	IF NOT Busy                                         	
	THEN                                                	
		IF ItpReadRParamsEx.bExecute                    	
		THEN                                            	
			Error											:=	ItpReadRParamsEx.bErr;
			ErrorId											:= ItpReadRParamsEx.nErrId;
		END_IF                          					
		IF NOT Execute                  					
		THEN                            	            	
			MemFnc											:= -1;
			ItpReadRParamsEx(bExecute := FALSE , sNciToPlc:= rNCIRef.NciToPlc);
		END_IF
	END_IF
	
	read													:= Busy;
END_METHOD

METHOD PUBLIC write : BOOL //Return value = TRUE if busy
//required parameter
//pAddr
//Index
//Count
//rNCIRef
VAR_INPUT
	Execute													:	BOOL;
END_VAR
	MemFnc 													:= FNC_WRITE;
	THIS^.Execute											:= Execute;

IF NOT __ISVALIDREF(rNCIRef) OR pAddr = 0 
THEN
	Busy													:= NOT Error;
	ErrorId													:= E_adsErr.DEVICE_INVALIDPARM;
	Error													:= TRUE;
	Done													:= FALSE;
	MemFnc													:= SEL(Execute , -1 ,MemFnc); 
	RETURN;
END_IF

	IF Execute
	THEN
		Error												:=	FALSE;
		ErrorId												:= 0;
		ItpWriteRParamsEx.bExecute 							:= TRUE;
	ELSIF NOT ItpWriteRParamsEx.bBusy   					
	THEN                                					
		Error												:=	FALSE;
		ErrorId												:= 0;
		ItpWriteRParamsEx.bExecute 							:= FALSE;

	END_IF

	ItpWriteRParamsEx(
		bExecute	:= ,
		pAddr		:= pAddr,
		nIndex		:= Index,
		nCount		:= Count,
		tTimeOut	:= ,
		sNciToPlc	:= rNCIRef.NciToPlc,
		bBusy		=> Busy,
		bErr		=> ,
		nErrId		=> );

	Done													:= NOT ItpWriteRParamsEx.bBusy
																AND NOT ItpWriteRParamsEx.bErr
																AND ItpWriteRParamsEx.bExecute;
                                        					
	IF NOT Busy
	THEN
		IF ItpWriteRParamsEx.bExecute
		THEN
			Error											:=	ItpWriteRParamsEx.bErr;
			ErrorId											:= ItpWriteRParamsEx.nErrId;
		END_IF                          					
		IF NOT Execute                  					
		THEN                            	
			MemFnc											:= -1;
			ItpWriteRParamsEx(bExecute := FALSE, sNciToPlc:= rNCIRef.NciToPlc);
		END_IF
	END_IF
	
	write													:= Busy;
END_METHOD

END_FUNCTION_BLOCK

// POUs/Motion/TF5100-NCI/NciChannel
{attribute 'no_check'}
FUNCTION_BLOCK NciChannel EXTENDS NCI_REF
VAR_INPUT
	Admin													:	NciAdmin;
	grp														:	NciGrp;
	Itp														:	NciItp;
	motion													:	NciMotion;
                        								   
	MFnc													: 	NciMFnc;
	RPara													:	NciReadWriteRParam;
                        								      
	Event													:	NciEventHandling;
                        	
END_VAR                 	
VAR_OUTPUT              	
	ErrHdl													:	ERROR_HDL;
END_VAR
VAR
END_VAR

	(* NCI Control											*)
	(********************************************************)

(********************************************************************************)
(* error event ctrl																*)
(********************************************************************************)
	Event(
		Enable			:= ,
		ConfirmTrig		:= NOT Errhdl.flag AND Event.Status.31 OR Admin.ResetAdmin,
		Name			:= ErrHdl.fnc,
		SourceId		:= (* Default *) ,
		rNci			:= THIS^,
		ErrorId			:= TO_UDINT(ErrHdl.Id),
		Status			=> );
		
	(* Reset FB errors by reset flag *)
	(* currently not in use, call _Resetting via state machine to reset Fb errors by setting Execute to FALSE 
	IF Admin.Reset
	THEN
		grp.Execute											:= grp.Execute AND NOT grp.Error;
		itp.Execute											:= itp.Execute AND NOT itp.Error;
		Motion.Execute										:= Motion.Execute AND NOT Motion.Error;
		RPara.Execute										:= RPara.Execute AND NOT RPara.Error;
	END_IF
	*)
	
(********************************************************************************)
(* work admin ctrl																*)
(********************************************************************************)
	admin(
		ResetAdmin					:= ,
		Enable					:= ,
		EStop					:= ,
		SingleBlockMode			:= , 
		InSingleBlockTrigNext	:= , 
		GrpCnfg					:= ,
		Override				:= ,
		SpindleOvr				:= ,	
		rNCIRef					:= THIS^,
		InGroup					=> ,
		Busy					=> ,
		Done					=> ,
		Error					=> ,
		ErrorID					=> ,
		ErrorText				=> );

(********************************************************************************)
(* work group ctrl																*)
(********************************************************************************)
	grp(
		Execute				:= ,
		Fnc					:= ,
		XAxisId				:= ,
		YAxisId				:= ,
		ZAxisId				:= ,
		Q1AxisId			:= ,
		Q2AxisId			:= ,
		Q3AxisId			:= ,
		Q4AxisId			:= ,
		Q5AxisId			:= ,
		AxisIndex			:= ,
		rNCIRef				:= THIS^, 
		Busy				=> ,
		Done				=> ,
		Error				=> ,
		ErrorID				=> ,
		ErrorText			=> );

(********************************************************************************)
(* work interpolation ctrl														*)
(********************************************************************************)
	Itp(
		Execute				:= ,
		Fnc					:= ,
		Prg					:= ,
		rTable				:= ,
		rNCIRef				:= THIS^,
		StartPrgAfterLoading:= , 
		LogFeederEntries	:= ,
		Busy				=> ,
		Done				=> ,
		Error				=> ,
		ErrorID				=> ,
		ErrorText			=> );


(********************************************************************************)
(* work motion ctrl																*)
(********************************************************************************)
	motion(
		Execute						:= ,
		Fnc							:= ,
		rNCIRef						:= THIS^,
		FNC_ESTOP					=> ,
		FNC_STEP_ON					=> ,
		FNC_ENABLE_FEEDER_BACKUP	=> ,
		FNC_DISABLE_FEEDER_BACKUP	=> ,
		FNC_RETRACE_FWD				=> ,
		FNC_RETRACE_BWD				=> ,
		Busy						=> ,
		Done						=> ,
		Error						=> ,
		ErrorId						=> ,
		ErrorText					=> );

(********************************************************************************)
(* work R rarameter ctrl														*)
(********************************************************************************)
	RPara(
		Execute						:= ,
		Fnc							:= ,
		pAddr						:= ,
		Index						:= ,
		Count						:= ,
		rNCIRef						:= THIS^,
		Done						=> ,
		Busy						=> ,
		Error						=> ,
		ErrorId						=> );

(********************************************************************************)
(* work M function  ctrl														*)
(********************************************************************************)
	MFnc(
		ConfirmHsk					:= ,
		FastMFuncReset				:= ,
		FastMFuncNo					:= ,
		rNCIRef						:= THIS^);

(********************************************************************************)
(* collect errors																*)
(********************************************************************************)
	IF Admin.Error
	THEN
		ErrHdl.flag											:= Admin.Error;
		ErrHdl.id											:= UDINT_TO_DINT(Admin.ErrorID);
		ErrHdl.fnc											:= 'NciAdmin';
		ErrHdl.text											:= Admin.ErrorText;
                        									
	ELSIF grp.Error     									
	THEN                									
		ErrHdl.flag											:= grp.Error;
		ErrHdl.id											:= UDINT_TO_DINT(grp.ErrorID);
		ErrHdl.fnc											:= 'NciGrp';
		ErrHdl.text											:= grp.ErrorText;
                        									
	ELSIF itp.Error     									
	THEN                									
		ErrHdl.flag											:= Itp.Error;
		ErrHdl.id											:= UDINT_TO_DINT(Itp.ErrorID);
		ErrHdl.fnc											:= 'NciItp';
		ErrHdl.text											:= Itp.ErrorText;
                        									
	ELSIF motion.Error  									
	THEN                									
		ErrHdl.flag											:= motion.Error;
		ErrHdl.id											:= UDINT_TO_DINT(motion.ErrorID);
		ErrHdl.fnc											:= 'NciMotion';
		ErrHdl.text											:= motion.ErrorText;
		
	ELSIF RPara.Error  									
	THEN                									
		ErrHdl.flag											:= RPara.Error;
		ErrHdl.id											:= UDINT_TO_DINT(RPara.ErrorID);
		ErrHdl.fnc											:= 'RPara';
		ErrHdl.text											:= CONCAT('Error RPara id: ',  UDINT_TO_STRING(RPara.Errorid));
	ELSE
		ErrHdl.Reset();
	END_IF
(******************************************************************************)

METHOD PUBLIC noAction : BOOL
VAR_INPUT
END_VAR
grp.Execute													:= FALSE;
itp.Execute													:= FALSE;
Motion.Execute												:= FALSE;
RPara.Execute												:= FALSE;

NoAction 													:= NOT Grp.Busy and not Itp.Busy and not Motion.Busy and not RPara.Busy;
END_METHOD

METHOD reset : Bool
VAR_INPUT
END_VAR
NoAction();
reset 			:= ErrHdl.flag OR Admin.reset(FALSE);
Event.confirm();
END_METHOD

END_FUNCTION_BLOCK

// POUs/Motion/TF511x-KIN/01_Main/KIN_REF
//Kinematic group ref - call ReadStatus cyclic
FUNCTION_BLOCK KIN_REF
VAR_INPUT
	PlcToNci										AT %Q*	:	PLCTONC_NCICHANNEL_REF;
END_VAR                     						
VAR_OUTPUT                  						
	NciToPlc										AT %I*	:	NCTOPLC_NCICHANNEL_REF;
                            						
	ChnOperationState										:	E_KINSTATUS := 0;
	CartesianModeON											:	BOOL := FALSE;
	                                					
(* ChnState ***************************)
	IsKinematicChn											:	BOOL := FALSE;
	                                					
	AxList													: ST_KinAxes;
END_VAR
VAR
END_VAR

;

METHOD PUBLIC readStatus : booL;
VAR_INPUT
END_VAR
(* Kin Channel State *********************************************************)
	F_KinGetAcsMcsAxisIds(AxList,NciToPlc);
	
	ChnOperationState 										:= TO_INT(F_KinGetChnOperationState(NciToPlc));

	CartesianModeON											:= NciToPlc.AcsAxisIDs[0] <> 0 AND NciToPlc.AcsAxisIDs[1] <> 0;
	
	IsKinematicChn											:= NciToPlc.ChnState.1;

	readStatus												:= TRUE;
(*****************************************************************************)
END_METHOD

END_FUNCTION_BLOCK

// POUs/Motion/TF511x-KIN/01_Main/KinAdmin
//Kinematic group administration - Enable/Disable/Reset group
//based on TF511x - Tc2_NcKinematicTransformation
//ACS - Axis coordinate system => Robot motors M1-Mx 
//MCS - Machine coordinate system >= Cartesian Axis X,Y,Z,Rx,Ry,Rz (A,B,C) 
FUNCTION_BLOCK KinAdmin
VAR_INPUT
	ResetTrig												:	BOOL := FALSE;
	Enable													:	BOOL := FALSE; (* TRUE = Build Group , FALSE = Reconfig Group *)
	Override												:	LREAL	:= 0.0;
	ItpChannelId 											: 	UDINT := 0; (* Bei 0 wirtd der ITP Kanal nicht resetet *)
	AxesList												: 	ST_KinAxes;
	rKINRef													:	REFERENCE TO KIN_REF := 0;
END_VAR
VAR_IN_OUT
END_VAR
VAR_OUTPUT
	Busy													:	BOOL;
	Done													:	BOOL;
	Error													:	BOOL;
{attribute 'displaymode':='hex'}
	ErrorId													:	UDINT;
	ErrorText												:	STRING(40);
END_VAR
VAR
(* cache **************************************************************************)
	MemDone													:	BOOL;
	MemFnc													:	INT := 1;
	                        								
(* MC-functonblock instances *******************************************************)
	ResetKinGroup											: 	FB_KinResetGroup ;
	ConfigKinGroup											:	FB_KinConfigGroup  ;

(* Dummy Speicher **********************************************************)
	OK 														: BOOL;
END_VAR

	(* Kinematic group administration										*)
	(************************************************************************)

(* aborting function-block call if pointer is not valid ****************************************)
IF NOT __ISVALIDREF(rKINRef) 
THEN
	Busy													:= NOT Error;
	ErrorId													:= E_AdsErr.DEVICE_INVALIDPARM;
	Error													:= TRUE;
	Done													:= FALSE;
	ErrorText												:= 'Reference to rKINRef invalid (0)';
	RETURN;
END_IF

(* reading axis-status from NCtoPLC-channel ***************************************************)
	rKINRef.readStatus();

(* accepting setvalue-barrier e.g. for hardware limit switch **********************************)
	rKINRef.PlcToNci.ChnAxesOvr 							:= LREAL_TO_DWORD(LIMIT(0.0,Override,100.0) * 10000.0 );

(* ctrl programm ******************************************************************************)
	ConfigKinGroup.bExecute									:=	NOT ConfigKinGroup.bBusy
																AND(
																Enable
																AND NOT ConfigKinGroup.bCartesianMode
																OR
																NOT Enable
																AND ConfigKinGroup.bCartesianMode);

	IF ConfigKinGroup.bExecute
	THEN
		ConfigKinGroup.bCartesianMode						:= Enable;
	END_IF

	ConfigKinGroup(
		bExecute		:= ,
		bCartesianMode	:= ,
		stAxesList		:= AxesList,
		stKinRefIn		:= rKinRef.NciToPlc,
		bBusy			=> ,
		bDone			=> ,
		bError			=> ,
		nErrorId		=> );

(* Reset Grp ****************************************************************)
	IF Memfnc < 0
	THEN
		IF ResetTrig
		THEN
			reset(Execute:= TRUE);
			MemFnc											:= 1;
		END_IF
	ELSIF NOT reset(Execute:= ResetTrig)
	THEN
		MemFnc												:= -1;
	END_IF

(******************************************************************************)
(* Ctrl Status 																					*)
(******************************************************************************)
	Busy						:= ResetKinGroup.bBusy OR ConfigKinGroup.bBusy;
	
	IF Busy
	THEN
		Error												:= FALSE;
		ErrorId												:= 0;
		ErrorText											:= '';
	ELSIF ConfigKinGroup.bError
	THEN
		Error												:= TRUE;
		ErrorId												:= ConfigKinGroup.nErrorID;
		ErrorText											:= CONCAT('ConfigKinGroup ErrorId: ', UDINT_TO_STRING(Errorid));
	ELSIF ResetKinGroup.bExecute
		AND ResetKinGroup.bError
	THEN
		Error												:= TRUE;
		ErrorId												:= ResetKinGroup.nErrorID;
		ErrorText											:= CONCAT('ResetKinGroup ErrorId: ', UDINT_TO_STRING(Errorid));
	ELSIF rKINRef.NciToPlc.ErrorCode <> 0
	THEN
		Error												:= TRUE;
		ErrorId												:= rKINRef.NciToPlc.ErrorCode;
		ErrorText											:= CONCAT('KIN Grp ErrorId: ', UDINT_TO_STRING(Errorid));
	ELSE
		Error												:= FALSE;
		ErrorId												:= 0;
		ErrorText											:= '';
	END_IF

	IF ResetKinGroup.bDone
		OR ConfigKinGroup.bDone
	THEN
		MemDone												:= TRUE;
	END_IF

	Done													:= NOT Busy AND MemDone;

	IF done
	THEN
		MemDone												:= FALSE;
	END_IF

(**************************************************************************************************)

METHOD PUBLIC reset : BOOL //Return value = TRUE if busy
//required parameter
//rKinRef
//ItpChannelId
//AxesList
VAR_INPUT
	Execute													:	BOOL;
END_VAR
IF NOT __ISVALIDREF(rKINRef) THEN
	Busy													:= NOT Error;
	ErrorId													:=E_AdsErr.DEVICE_INVALIDPARM;
	Error													:= TRUE;
	Done													:= FALSE;
	ErrorText												:= 'Reference to rKINRef  invalid (0)';
	RETURN;
END_IF

	IF Execute
	THEN
		Error												:=	FALSE;
		ErrorId												:= 0;
		ResetKinGroup.bExecute 								:= rKinRef.NciToPlc.ErrorCode <> 0;
	ELSIF NOT ResetKinGroup.bBusy
	THEN
		Error												:=	FALSE;
		ErrorId												:= 0;
		ResetKinGroup.bExecute 								:= FALSE;

	END_IF

	ResetKinGroup(
		bExecute		:= ,
		nItpChannelId	:= ItpChannelId,
		stKinRefIn		:= rKinRef.NciToPlc,
		stAxesList		:= AxesList,
		bBusy			=> Busy,
		bDone			=> ,
		bError			=> ,
		nErrorId		=> );

	Done													:= NOT ResetKinGroup.bBusy
																AND NOT ResetKinGroup.bError
																AND ResetKinGroup.bExecute;

	IF NOT Busy
	THEN
		IF ResetKinGroup.bExecute
		THEN
			Error											:=	ResetKinGroup.bError;
			ErrorId											:= ResetKinGroup.nErrorId;
			ErrorText										:= SEL(Error , '' ,  CONCAT('Error ResetKinGroup id: ',  UDINT_TO_STRING(Errorid)));
		END_IF
		IF NOT Execute
		THEN
			MemFnc											:= -1 ;
			ResetKinGroup(	bExecute := FALSE, 
							stKinRefIn := rKinRef.NciToPlc, 
							stAxesList := AxesList);
		END_IF
	END_IF
	
	reset													:= Busy;
END_METHOD

END_FUNCTION_BLOCK

// POUs/Motion/TF511x-KIN/02_Options/KinLockUnlockTrafoParam
//Lock or Unlock kinematic group parameter
FUNCTION_BLOCK KinLockUnlockTrafoParam
VAR_INPUT
	Execute													:	BOOL	:= FALSE;
	Lock													:	BOOL 	:= TRUE;
   	oidTrafo												:	UDINT;
END_VAR                     								
VAR_OUTPUT                  								
	Busy													:	BOOL	:= FALSE;
	Done													:	BOOL	:= FALSE;
	Error													:	BOOL	:= FALSE;
	ErrorId													:	UDINT	:= 0;
END_VAR                     								
VAR                         	
	State													:	UDINT	:= 0;
	ADSWRITE												:	ADSWRITE;
END_VAR

CASE State OF
0:
	Done													:= FALSE;
	Error													:= FALSE;
	ErrorId													:= 0;
	Busy 													:= FALSE;
	
	IF Execute THEN
		AdsWrite(WRITE := FALSE);
		AdsWrite(
			NETID		:='',
			PORT		:= 10,
			IDXGRP		:=oidTrafo,
			IDXOFFS		:=SEL(Lock, 16#05030210, 16#0503020F),
			LEN			:= 0,
			SRCADDR		:=0 ,
			WRITE		:= TRUE,
			TMOUT		:= DEFAULT_ADS_TIMEOUT,
			BUSY		=> ,
			ERR			=> ,
			ERRID		=> );

		Busy												:= TRUE;
		State												:= 10;
	END_IF
10:
	AdsWrite(
		TMOUT	:= DEFAULT_ADS_TIMEOUT,
		BUSY	=>,
		ERR		=>Error,
		ERRID	=>ErrorId);
		
	IF NOT AdsWrite.BUSY 
	THEN
		IF NOT AdsWrite.ERR 
		THEN
			Done											:= TRUE;
		END_IF
		IF NOT Execute THEN
			State											:= 0;
		ELSE
			State											:= 20;
		END_IF
		AdsWrite(WRITE:=FALSE);
	END_IF
20:
	Busy													:= FALSE;
	IF NOT Execute THEN
		State												:= 0;
	END_IF

END_CASE

END_FUNCTION_BLOCK

// POUs/Motion/TF511x-KIN/02_Options/KinWriteToolTrafoParam
{attribute 'hide'}
(*==============================================================================*)
(* Name:			KIN_WriteToolTrafoParam							  	 		*)
(* Desc:			THIS IS NOT A RELEASED IMPLEMENTATION AND    				*)
(*  	           	SUBJECT TO CHANGE                            				*)
(*     			 															    *)
(* Author:	 	DS																*)
(* Date:							     										*)
(*==============================================================================*)
FUNCTION_BLOCK KinWriteToolTrafoParam
VAR_INPUT
	Execute													:	BOOL	:= FALSE;
   	oidTrafo												:	UDINT;
	ToolX													:	LREAL := 0.0;
	ToolY													:	LREAL := 0.0;
	ToolZ													:	LREAL := 0.0;
END_VAR                     								
VAR_OUTPUT                  								
	Busy													:	BOOL	:= FALSE;
	Done													:	BOOL	:= FALSE;
	Error													:	BOOL	:= FALSE;
	ErrorId													:	UDINT	:= 0;
END_VAR
VAR
	State													:	UDINT	:= 0;
	ADSWRITE												:ADSWRITE;
END_VAR

CASE State OF
0:
	Done													:= FALSE;
	Busy 													:= FALSE;
	Error													:= FALSE;
	ErrorId													:= 0;
	IF Execute 
	THEN
		AdsWrite(WRITE := FALSE);
		AdsWrite(
			NETID	:='',
			PORT	:= 10,
			IDXGRP	:=oidTrafo,
			IDXOFFS	:=SEL(FALSE (* Lock *), 16#05030210, 16#0503020F),
			LEN		:= 0,
			SRCADDR	:=0 ,
			WRITE	:= TRUE,
			TMOUT	:= DEFAULT_ADS_TIMEOUT,
			BUSY	=> ,
			ERR		=> ,
			ERRID	=> );

		Busy												:= TRUE;
		State												:= 1;
	END_IF

1:
	AdsWrite(
		TMOUT	:= DEFAULT_ADS_TIMEOUT,
		BUSY	=>,
		ERR		=>Error,
		ERRID	=>ErrorId);
		
	IF NOT AdsWrite.BUSY 
	THEN
		AdsWrite(WRITE:=FALSE);
			
		IF NOT AdsWrite.ERR 
		THEN
			AdsWrite( (* Write Tool X *)
				NETID	:= '',
				PORT	:= 10,
				IDXGRP	:= oidTrafo, 				(*OID 	Tool trafo*)
				IDXOFFS	:= 16#05010020, 			(*PTCID	Tool Trafo Parameter*)
				LEN		:= SIZEOF(ToolX),
				SRCADDR	:= ADR(ToolX),
				TMOUT	:= DEFAULT_ADS_TIMEOUT,
				WRITE 	:= TRUE,
				BUSY	=> ,
				ERR		=> ,
				ERRID	=> );
	

			State											:= 10;
		ELSE
			IF NOT Execute
			THEN
				State										:= 0;
			ELSE
				State										:= 99;
			END_IF
		END_IF
	END_IF

10:
	AdsWrite(
		TMOUT	:= DEFAULT_ADS_TIMEOUT,
		BUSY	=>,
		ERR		=>Error,
		ERRID	=>ErrorId);
		
	IF NOT AdsWrite.BUSY 
	THEN
		AdsWrite(WRITE:=FALSE);
		
		IF NOT AdsWrite.ERR 
		THEN
			AdsWrite( 								(* Write Tool Y *)
				NETID	:= '',
				PORT	:= 10,
				IDXGRP	:= oidTrafo, 				(*OID 	Tool trafo*)
				IDXOFFS	:= 16#05010021, 			(*PTCID	Tool Trafo Parameter*)
				LEN		:= SIZEOF(ToolY),
				SRCADDR	:= ADR(ToolY),
				TMOUT	:= DEFAULT_ADS_TIMEOUT,
				WRITE	:= TRUE,
				BUSY	=> ,
				ERR		=> ,
				ERRID	=> );

			State											:= 20;
		ELSE
			State											:= 90;
		END_IF
	END_IF

20:
	AdsWrite(
		TMOUT	:= DEFAULT_ADS_TIMEOUT,
		BUSY	=>,
		ERR		=>Error,
		ERRID	=>ErrorId);

	IF NOT AdsWrite.BUSY 
	THEN
		AdsWrite(WRITE:=FALSE);
		
	IF NOT AdsWrite.ERR 
	THEN
			AdsWrite( 								(* Write Tool Z *)
				NETID	:= '',
				PORT	:= 10,
				IDXGRP	:= oidTrafo, 				(*OID 	Tool trafo*)
				IDXOFFS	:= 16#05010022, 			(*PTCID	Tool Trafo Parameter*)
				LEN		:= SIZEOF(ToolZ),
				SRCADDR	:= ADR(ToolZ),
				TMOUT	:= DEFAULT_ADS_TIMEOUT,
				WRITE 	:= TRUE,
				BUSY	=> ,
				ERR		=> ,
				ERRID	=> );

			State											:= 60;
		ELSE            									
			State											:= 90;
		END_IF
	END_IF

60:
	AdsWrite(
		TMOUT	:= DEFAULT_ADS_TIMEOUT,
		BUSY	=>,
		ERR		=>Error,
		ERRID	=>ErrorId);

	IF NOT AdsWrite.BUSY 
	THEN
		State												:= 90;
		AdsWrite(WRITE:=FALSE);
	END_IF


90: (* Start Lock-Param *)
	AdsWrite(
		NETID	:='',
		PORT	:= 10,
		IDXGRP	:=oidTrafo,
		IDXOFFS	:=SEL(TRUE (* Lock *), 16#05030210, 16#0503020F),
		LEN		:= 0,
		SRCADDR	:=0 ,
		WRITE	:= TRUE,
		TMOUT	:= DEFAULT_ADS_TIMEOUT,
		BUSY	=> ,
		ERR		=> ,
		ERRID	=> );

	State													:= 91;

91:
	AdsWrite(
		TMOUT	:= DEFAULT_ADS_TIMEOUT,
		BUSY	=>,
		ERR		=>,
		ERRID	=>);

	IF NOT AdsWrite.BUSY 
	THEN
		Busy 												:= FALSE;
		IF NOT AdsWrite.ERR 
		THEN
			Done											:= NOT Error;
		ELSIF NOT Error
		THEN
			Error 											:= AdsWrite.ERR;
			ErrorId 										:= AdsWrite.ERRID;
		END_IF
		IF NOT Execute 
		THEN
			State											:= 0;
		ELSE        										
			State											:= 99;
		END_IF
		AdsWrite(WRITE:=FALSE);
	END_IF

99:
	Busy													:= FALSE;
	IF NOT Execute THEN
		State												:= 0;
	END_IF

END_CASE

END_FUNCTION_BLOCK

// POUs/Motion/TF511x-KIN/02_Options/KinWriteUCSTrafoParam
{attribute 'hide'}
(*==============================================================================*)
(* Name:			KIN_WriteUCSTrafoParam							  	 		*)
(* Desc:			THIS IS NOT A RELEASED IMPLEMENTATION AND    				*)
(*  	           	SUBJECT TO CHANGE                            				*)
(*     			 															    *)
(* Author:	 	DS																*)
(* Date:							     										*)
(*==============================================================================*)
FUNCTION_BLOCK KinWriteUCSTrafoParam
VAR_INPUT
	Execute													:	BOOL	:= FALSE;
   oidTrafo													:	UDINT;
	vTranslation 											:	VECTOR;
 	vRotation 												:	VECTOR;
END_VAR
VAR_OUTPUT
	Busy													:	BOOL	:= FALSE;
	Done													:	BOOL	:= FALSE;
	Error													:	BOOL	:= FALSE;
	ErrorId													:	UDINT	:= 0;
END_VAR
VAR
	State													:	UDINT	:= 0;
	ADSWRITE												:ADSWRITE;
END_VAR

CASE State OF
0:
	Done													:= FALSE;
	Busy													:= FALSE;
	Error													:= FALSE;
	ErrorId													:= 0;
	IF Execute 
	THEN
		AdsWrite(WRITE := FALSE);
		AdsWrite(
			NETID	:='',
			PORT	:= 10,
			IDXGRP	:=oidTrafo,
			IDXOFFS	:=SEL(FALSE (* Lock *), 16#05030210, 16#0503020F),
			LEN		:= 0,
			SRCADDR	:=0 ,
			WRITE	:= TRUE,
			TMOUT	:= DEFAULT_ADS_TIMEOUT,
			BUSY	=> ,
			ERR		=> ,
			ERRID	=> );

		Busy												:= TRUE;
		State												:= 1;
	END_IF

1: (* Start Translation X *)
	AdsWrite(
		TMOUT	:= DEFAULT_ADS_TIMEOUT,
		BUSY	=>,
		ERR		=>Error,
		ERRID	=>ErrorId);
		
	IF NOT AdsWrite.BUSY 
	THEN
		AdsWrite(WRITE:=FALSE);
		IF NOT AdsWrite.ERR 
		THEN
			AdsWrite(
				NETID	:= '',
				PORT	:= 10,
				IDXGRP	:= oidTrafo,
				IDXOFFS	:= 16#05010020,
				LEN		:= SIZEOF(vTranslation.m[1]),
				SRCADDR	:= ADR(vTranslation.m[1]),
				TMOUT	:= DEFAULT_ADS_TIMEOUT,
				WRITE 	:= TRUE,
				BUSY	=> ,
				ERR		=> ,
				ERRID	=> );

			State											:= 10;
		ELSE (* Error unlock Param *)
			IF NOT Execute 
			THEN
				State										:= 0;
			ELSE
				State										:= 99;
			END_IF
		END_IF
	END_IF

10: (* Translation Y *)
	AdsWrite(
		TMOUT	:= DEFAULT_ADS_TIMEOUT,
		BUSY	=>,
		ERR		=>Error,
		ERRID	=>ErrorId);
		
	IF NOT AdsWrite.BUSY 
	THEN
		AdsWrite(WRITE:=FALSE);
		
		IF NOT AdsWrite.ERR 
		THEN
			AdsWrite(
				NETID	:= '',
				PORT	:= 10,
				IDXGRP	:= oidTrafo,
				IDXOFFS	:= 16#05010021,
				LEN		:= SIZEOF(vTranslation.m[2]),
				SRCADDR	:= ADR(vTranslation.m[2]),
				TMOUT	:= DEFAULT_ADS_TIMEOUT,
				WRITE 	:= TRUE,
				BUSY	=> ,
				ERR		=> ,
				ERRID	=> );

			State											:= 20;
		ELSE            									
			State											:= 90;
		END_IF

	END_IF

20: (* Translation Z *)
	AdsWrite(
		TMOUT	:= DEFAULT_ADS_TIMEOUT,
		BUSY	=>,
		ERR		=>Error,
		ERRID	=>ErrorId);

	IF NOT AdsWrite.BUSY 
	THEN
		AdsWrite(WRITE:=FALSE);
		IF NOT AdsWrite.ERR 
		THEN
			AdsWrite(
				NETID	:= '',
				PORT	:= 10,
				IDXGRP	:= oidTrafo,
				IDXOFFS	:= 16#05010022,
				LEN		:= SIZEOF(vTranslation.m[3]),
				SRCADDR	:= ADR(vTranslation.m[3]),
				TMOUT	:= DEFAULT_ADS_TIMEOUT,
				WRITE 	:= TRUE,
				BUSY	=> ,
				ERR		=> ,
				ERRID	=> );

			State											:= 30;
		ELSE
			State											:= 90;
		END_IF

	END_IF

30: (* Roation X *)
	AdsWrite(
		TMOUT	:= DEFAULT_ADS_TIMEOUT,
		BUSY	=>,
		ERR		=>Error,
		ERRID	=>ErrorId);

	IF NOT AdsWrite.BUSY 
	THEN
		AdsWrite(WRITE:=FALSE);
		IF NOT AdsWrite.ERR 
		THEN
			AdsWrite(
				NETID	:= '',
				PORT	:= 10,
				IDXGRP	:= oidTrafo,
				IDXOFFS	:= 16#05010060,
				LEN		:= SIZEOF(VRotation.m[1]),
				SRCADDR	:= ADR(VRotation.m[1]),
				TMOUT	:= DEFAULT_ADS_TIMEOUT,
				WRITE 	:= TRUE,
				BUSY	=> ,
				ERR		=> ,
				ERRID	=> );

			State											:= 40;
		ELSE
			State											:= 90;
		END_IF
	END_IF

40: (* Roation Y *)
	AdsWrite(
		TMOUT	:= DEFAULT_ADS_TIMEOUT,
		BUSY	=>,
		ERR		=>Error,
		ERRID	=>ErrorId);

	IF NOT AdsWrite.BUSY 
	THEN
		AdsWrite(WRITE:=FALSE);
		IF NOT AdsWrite.ERR 
		THEN
			AdsWrite(
				NETID	:= '',
				PORT	:= 10,
				IDXGRP	:= oidTrafo,
				IDXOFFS	:= 16#05010061,
				LEN		:= SIZEOF(VRotation.m[2]),
				SRCADDR	:= ADR(VRotation.m[2]),
				TMOUT	:= DEFAULT_ADS_TIMEOUT,
				WRITE 	:= TRUE,
				BUSY	=> ,
				ERR		=> ,
				ERRID	=> );
			State											:= 50;
		ELSE            									
			State											:= 90;
		END_IF

	END_IF

50: (* Roation Z *)
	AdsWrite(
		TMOUT	:= DEFAULT_ADS_TIMEOUT,
		BUSY	=>,
		ERR		=>Error,
		ERRID	=>ErrorId);

	IF NOT AdsWrite.BUSY 
	THEN
		AdsWrite(WRITE:=FALSE);
		IF NOT AdsWrite.ERR 
		THEN
			AdsWrite(
				NETID	:= '',
				PORT	:= 10,
				IDXGRP	:= oidTrafo,
				IDXOFFS	:= 16#05010062,
				LEN		:= SIZEOF(VRotation.m[3]),
				SRCADDR	:= ADR(VRotation.m[3]),
				TMOUT	:= DEFAULT_ADS_TIMEOUT,
				WRITE 	:= TRUE,
				BUSY	=> ,
				ERR		=> ,
				ERRID	=> );

			State											:= 60;
		ELSE            									
			State											:= 90;
		END_IF
	END_IF

60:
	AdsWrite(
		TMOUT	:= DEFAULT_ADS_TIMEOUT,
		BUSY	=>,
		ERR		=>Error,
		ERRID	=>ErrorId);

	IF NOT AdsWrite.BUSY 
	THEN
		State												:= 90;
		AdsWrite(WRITE:=FALSE);
	END_IF

90: (* Start Lock-Param *)
	AdsWrite(
		NETID	:='',
		PORT	:= 10,
		IDXGRP	:=oidTrafo,
		IDXOFFS	:=SEL(TRUE (* Lock *), 16#05030210, 16#0503020F),
		LEN		:= 0,
		SRCADDR	:=0 ,
		WRITE	:= TRUE,
		TMOUT	:= DEFAULT_ADS_TIMEOUT,
		BUSY	=> ,
		ERR		=> ,
		ERRID	=> );

	State													:= 91;

91:
	AdsWrite(
		TMOUT	:= DEFAULT_ADS_TIMEOUT,
		BUSY	=>,
		ERR		=>,
		ERRID	=>);

	IF NOT AdsWrite.BUSY 
	THEN
		Busy 												:= FALSE;
		IF NOT AdsWrite.ERR 
		THEN
			Done											:= NOT Error;
		ELSIF NOT Error
		THEN
			Error 											:= AdsWrite.ERR;
			ErrorId 										:= AdsWrite.ERRID;
		END_IF
		IF NOT Execute 
		THEN
			State											:= 0;
		ELSE        										
			State											:= 99;
		END_IF
		AdsWrite(WRITE:=FALSE);
	END_IF

99:
	Busy 													:= FALSE;
	IF NOT Execute 
	THEN
		State												:= 0;
	END_IF

END_CASE

END_FUNCTION_BLOCK

// POUs/Motion/TF511x-KIN/03_DUTs/Positions/KIN_POSITIONS
{attribute 'no_check'}
FUNCTION_BLOCK KIN_POSITIONS 
VAR_INPUT
	Valid													:	BOOL ;
	MCS														:	KIN_POSITIONS_MCS_DUT; //Values as union
END_VAR
VAR_OUTPUT
END_VAR
VAR
END_VAR

;

METHOD PUBLIC copy : BOOL //Return value = TRUE if execution finished
VAR_IN_OUT
	Source													:	KIN_POSITIONS;
END_VAR
	Valid													:= Source.Valid;
	MCS														:= Source.MCS;
	copy													:= TRUE;
END_METHOD

METHOD PUBLIC delete : BOOL //Return value = TRUE if execution finished - Valid bit will not change
VAR_INPUT
END_VAR
	MCS.A													:= 0.0;
	MCS.B													:= 0.0;
	MCS.C													:= 0.0;
	MCS.X													:= 0.0;
	MCS.Y													:= 0.0;
	MCS.Z													:= 0.0;
	MCS.Q1													:= 0.0;
	MCS.Q2													:= 0.0;
	
	delete													:= TRUE;
END_METHOD

METHOD PUBLIC isInPos : BOOL //Return value = TRUE if axes are within window of checkPos values
VAR_IN_OUT
	CheckPos												:	KIN_POSITIONS_MCS_DUT;
	Window													:	KIN_POSITIONS_MCS_DUT;
END_VAR             										
VAR CONSTANT        										
END_VAR
IsInPos 														:= IsInPosXYZ(CheckPos,Window) AND IsInPosABC(CheckPos,Window);
END_METHOD

METHOD PUBLIC isInPosABC : BOOL //Return value = TRUE if axes are within window of checkPos values
VAR_IN_OUT
	CheckPos												:	KIN_POSITIONS_MCS_DUT;
	Window													:	KIN_POSITIONS_MCS_DUT;
END_VAR                 									
VAR CONSTANT            									
END_VAR
isInPosABC												 	:= CAM(CheckPos.A, MCS.A ,Window.A)
																AND CAM(CheckPos.B, MCS.B ,Window.B)
																AND CAM(CheckPos.C, MCS.C ,Window.C);
END_METHOD

METHOD PUBLIC isInPosByAxisNo : BOOL //Return value = TRUE selected axis is within window of checkPos values
VAR_INPUT
	No					:	INT;
END_VAR
VAR_IN_OUT
	CheckPos			:	KIN_POSITIONS_MCS_DUT;
	Window				:	KIN_POSITIONS_MCS_DUT;
END_VAR
isInPosByAxisNo													:= (CAM(CheckPos.X, MCS.X ,Window.X) OR No <> 1)
																AND (CAM(CheckPos.Y, MCS.Y ,Window.Y) OR No <> 2)
																AND (CAM(CheckPos.Z, MCS.Z ,Window.Z) OR No <> 3)
																AND (CAM(CheckPos.A, MCS.A ,Window.A) OR No <> 4)
																AND (CAM(CheckPos.B, MCS.B ,Window.B) OR No <> 5)
																AND (CAM(CheckPos.C, MCS.C ,Window.C) OR No <> 6)
																AND (CAM(CheckPos.Q1, MCS.Q1 ,Window.Q1) OR No <> 7)
																AND (CAM(CheckPos.Q2, MCS.Q2 ,Window.Q2) OR No <> 8);
END_METHOD

METHOD PUBLIC isInPosExt : BOOL //Return value = TRUE if axes are within window of checkPos values
VAR_INPUT
{attribute 'displaymode':='binary'}
	Config													:	DWORD; //Select value to be checked by bis mask .0=X or A1, .1=Y or A2, .3=Y or A3.....
END_VAR
VAR_IN_OUT
	CheckPos												:	KIN_POSITIONS_MCS_DUT;
	Window													:	KIN_POSITIONS_MCS_DUT;
END_VAR                 									
VAR CONSTANT            									
END_VAR
isInPosExt													:= (CAM(CheckPos.X, MCS.X ,Window.X) OR NOT Config.0)
																AND (CAM(CheckPos.Y, MCS.Y ,Window.Y) OR NOT Config.1)
																AND (CAM(CheckPos.Z, MCS.Z ,Window.Z) OR NOT Config.2)
																AND (CAM(CheckPos.A, MCS.A ,Window.A) OR NOT Config.3)
																AND (CAM(CheckPos.B, MCS.B ,Window.B) OR NOT Config.4)
																AND (CAM(CheckPos.C, MCS.C ,Window.C) OR NOT Config.5)
																AND (CAM(CheckPos.Q1, MCS.Q1 ,Window.Q1) OR NOT Config.6)
																AND (CAM(CheckPos.Q2, MCS.Q2 ,Window.Q2) OR NOT Config.7);
END_METHOD

METHOD PUBLIC isInPosXYZ : BOOL //Return value = TRUE if axes are within window of checkPos values
VAR_IN_OUT
	CheckPos												:	KIN_POSITIONS_MCS_DUT;
	Window													:	KIN_POSITIONS_MCS_DUT;
END_VAR                 									
VAR CONSTANT            									
END_VAR
IsInPosXYZ												 	:= CAM(CheckPos.X, MCS.X ,Window.X)
																AND CAM(CheckPos.Y, MCS.Y ,Window.Y)
																AND CAM(CheckPos.Z, MCS.Z ,Window.Z);
END_METHOD

METHOD PUBLIC reset : BOOL //Delete data and reset valid , TRUE if execution finished
VAR_INPUT
END_VAR
Delete(); 
Valid														:= FALSE;
reset														:= TRUE;
END_METHOD

END_FUNCTION_BLOCK

// POUs/Motion/TF511x-KIN/03_DUTs/Trafo/KIN_CALCTRAFO_AXPOS_PARAM
FUNCTION_BLOCK KIN_CALCTRAFO_AXPOS_PARAM
VAR_INPUT
	In														: 	ARRAY[1..8] OF LREAL;
	Out														: 	ARRAY[1..8] OF LREAL;
	MetaInfoIn												:	U_KinMetaInfo;
	MetaInfoOut												:	U_KinMetaInfo;
END_VAR
VAR_OUTPUT
END_VAR
VAR
END_VAR

METHOD delete : BOOL
VAR_INPUT
END_VAR
MEMSET(ADR(In),0,SIZEOF(In));
MEMSET(ADR(Out),0,SIZEOF(Out));
delete	:= TRUE;
END_METHOD

END_FUNCTION_BLOCK

// POUs/Motion/TF511x-KIN/03_DUTs/Trafo/KIN_STATE_OBSERVER_OID_PARAM
{attribute 'hide'}
FUNCTION_BLOCK KIN_STATE_OBSERVER_OID_PARAM
VAR_INPUT
	oid														:	UDINT := 0; (* Scara State Observer OID *)
	TooltrafoOID											:	UDINT := 0; (* ToolTrafoOID *)
	NextTrafoOID											:	UDINT := 0; (*StaticTrafoOID *)

END_VAR
VAR_OUTPUT

END_VAR
VAR
END_VAR

;

METHOD delete : BOOL
VAR_INPUT
END_VAR
	oid														:= 0;
	TooltrafoOID											:= 0;
	NextTrafoOID											:= 0;
delete	:= TRUE;
END_METHOD

END_FUNCTION_BLOCK

// POUs/Motion/TF511x-KIN/03_DUTs/Trafo/KIN_STATICTRAFO_PARAM
{attribute 'hide'}
FUNCTION_BLOCK KIN_STATICTRAFO_PARAM
VAR_INPUT
	oid														:	UDINT := 0;
	TranslationX											:	LREAL := 0.0;
	TranslationY											:	LREAL := 0.0;
	TranslationZ											:	LREAL := 0.0;
                            								
	Rotation												: LREAL := 0.0;
	RotationAxis											: INT := 2;

END_VAR
VAR_OUTPUT

END_VAR
VAR
END_VAR

;

METHOD delete : BOOL
VAR_INPUT
END_VAR
	oid														:= 0;
	TranslationX											:= 0.0;
	TranslationY											:= 0.0;
	TranslationZ											:= 0.0;
                            								
	Rotation												:= 0.0;
	RotationAxis											:= 2;
delete	:= TRUE;
END_METHOD

END_FUNCTION_BLOCK

// POUs/Motion/TF511x-KIN/03_DUTs/Trafo/KIN_TOOLTRAFO_PARAM
{attribute 'hide'}
FUNCTION_BLOCK KIN_TOOLTRAFO_PARAM
VAR_INPUT
	oid														:	UDINT := 0;
	dx														: 	LREAL := 0.0;  (* Default Tooldata at WOS *)
	dy														: 	LREAL := 0.0;  (* Default Tooldata at WOS *)
	dz														:	LREAL := 0.0;  (* Default Tooldata at WOS *)

END_VAR
VAR_OUTPUT

END_VAR
VAR
END_VAR

;

METHOD delete : BOOL
VAR_INPUT
END_VAR
	oid														:= 0;
	dx														:= 0.0;  (* Default Tooldata at WOS *)
	dy														:= 0.0;  (* Default Tooldata at WOS *)
	dz														:= 0.0;  (* Default Tooldata at WOS *)
delete	:= TRUE;
END_METHOD

END_FUNCTION_BLOCK

// POUs/Motion/TF511x-KIN/KinChannel
FUNCTION_BLOCK KinChannel EXTENDS KIN_REF
VAR_INPUT
	Admin													:	KinAdmin;
END_VAR
VAR_OUTPUT
END_VAR
VAR
END_VAR

(* Kinematic Ctrl 										*)
(********************************************************)

(* work IO ********************************************************************)
(*	IO(); *)
	
(****************************************************************************)
(* Kinematic group control													*)
(****************************************************************************)
	Admin(
		ResetTrig			:= ,
		Enable			:= ,
		Override		:= ,
		ItpChannelId	:= ,
		AxesList		:= ,
		rKINRef			:= THIS^,
		Busy			=> ,
		Done			=> ,
		Error			=> ,
		ErrorId			=> );
(****************************************************************************)

END_FUNCTION_BLOCK

// POUs/Motion/VALUE_3D
{attribute 'no_check'}
FUNCTION_BLOCK VALUE_3D
VAR_INPUT                                                            
	Valid													:	BOOL ;
	X														:	LREAL;
	Y														:	LREAL;
	Z														:	LREAL;
END_VAR
VAR_OUTPUT
END_VAR
VAR
END_VAR

;

METHOD PUBLIC copy : BOOL //Return value = TRUE if execution finished
VAR_IN_OUT
	Source													:	VALUE_3D;
END_VAR
	Valid													:= Source.Valid;
	X														:= Source.X;
	Y														:= Source.Y;
	Z														:= Source.Z;
	copy													:= TRUE;
END_METHOD

METHOD PUBLIC delete : BOOL //Return value = TRUE if execution finished - Valid bit will not change
VAR_INPUT
END_VAR
	X					 									:= 0.0;	
	Y					 									:= 0.0;	
	Z					 									:= 0.0;	
	delete													:= TRUE;
END_METHOD

METHOD PUBLIC InPos : BOOL //Return value = TRUE axes is within window of checkPos values
VAR_IN_OUT
	CheckPos												:	VALUE_3D;
	Window													:	VALUE_3D;
END_VAR
InPos														:= CAM(CheckPos.X, X ,Window.X)
																AND CAM(CheckPos.Y, Y ,Window.Y)
																AND CAM(CheckPos.Z, Z ,Window.Z);
END_METHOD

METHOD PUBLIC InPosByAxisNo : BOOL //Return value = TRUE selected axis is within window of checkPos values
VAR_INPUT
	No					:	INT;
END_VAR
VAR_IN_OUT
	CheckPos			:	VALUE_3D;
	Window				:	VALUE_3D;
END_VAR
InPosByAxisNo													:= (CAM(CheckPos.X, X ,Window.X) OR No <> 1)
																AND (CAM(CheckPos.Y, Y ,Window.Y) OR No <> 2)
																AND (CAM(CheckPos.Z, Z ,Window.Z) OR No <> 3);
END_METHOD

METHOD PUBLIC InPosXY : BOOL //Return value = TRUE if axes are within window of checkPos values
VAR_IN_OUT
	CheckPos			:	VALUE_3D;
	Window				:	VALUE_3D;
END_VAR
InPosXY 													:= CAM(CheckPos.X, X ,Window.X)
																AND CAM(CheckPos.Y, Y ,Window.Y);
END_METHOD

METHOD PUBLIC InPosXZ : BOOL //Return value = TRUE if axes are within window of checkPos values
VAR_IN_OUT
	CheckPos			:	VALUE_3D;
	Window				:	VALUE_3D;
	
END_VAR
InPosXZ														:= CAM(CheckPos.X, X ,Window.X)
																AND CAM(CheckPos.Z, Z ,Window.Z);
END_METHOD

METHOD PUBLIC InPosYZ : BOOL //Return value = TRUE if axes are within window of checkPos values
VAR_IN_OUT
	CheckPos			:	VALUE_3D;
	Window				:	VALUE_3D;
	
END_VAR
InPosYZ													:= CAM(CheckPos.Y, Y ,Window.Y)
																AND CAM(CheckPos.Z, Z ,Window.Z);
END_METHOD

METHOD PUBLIC reset : BOOL //Delete data and reset valid , TRUE if execution finished
VAR_INPUT
END_VAR
Delete();
Valid														:= FALSE;
reset														:= TRUE;
END_METHOD

END_FUNCTION_BLOCK

// POUs/Motion/VALUE_6D
{attribute 'no_check'}
FUNCTION_BLOCK VALUE_6D 
VAR_INPUT
	Valid													:	BOOL ;
	X														:	LREAL;
	Y														:	LREAL;
	Z														:	LREAL;
	A														:		LREAL; //Rx
	B														:		LREAL; //Ry
	C														:		LREAL; //Rz	
END_VAR
VAR_OUTPUT
END_VAR
VAR
END_VAR

;

METHOD PUBLIC copy : BOOL //Return value = TRUE if execution finished
VAR_IN_OUT
	Source													:	VALUE_6D;
END_VAR
	Valid													:= Source.Valid;
	X														:= Source.X;
	Y														:= Source.Y;
	Z														:= Source.Z;
	A														:= Source.A;
	B														:= Source.B;
	C														:= Source.C;
	copy													:= TRUE;
END_METHOD

METHOD PUBLIC delete : BOOL //Return value = TRUE if execution finished - Valid bit will not change
VAR_INPUT
END_VAR
	X					 									:= 0.0;	
	Y					 									:= 0.0;	
	Z					 									:= 0.0;	
	A						 								:= 0.0;	
	B						 								:= 0.0;	
	C						 								:= 0.0;	
	delete													:= TRUE;
END_METHOD

METHOD PUBLIC inPos : BOOL //Return value = TRUE if axes are within window of checkPos values
VAR_IN_OUT
	CheckPos												:	VALUE_6D;
	Window													:	VALUE_6D;
END_VAR             										
VAR CONSTANT        										
END_VAR
InPos 														:= CAM(CheckPos.X, X, Window.X)
																AND CAM(CheckPos.Y, Y ,Window.Y)
																AND CAM(CheckPos.Z, Z,Window.Z)
																AND CAM(CheckPos.A, A, Window.A)
																AND CAM(CheckPos.B, B ,Window.B)
																AND CAM(CheckPos.C, C,Window.C);
END_METHOD

METHOD PUBLIC InPosABC : BOOL //Return value = TRUE if axes are within window of checkPos values
VAR_IN_OUT
	CheckPos												:	VALUE_6D;
	Window													:	VALUE_6D;
END_VAR                 									
VAR CONSTANT            									
END_VAR
InPosABC												 	:= CAM(CheckPos.A, A ,Window.A)
																AND CAM(CheckPos.B, B ,Window.B)
																AND CAM(CheckPos.C, C ,Window.C);
END_METHOD

METHOD PUBLIC InPosAC : BOOL //Return value = TRUE if axes are within window of checkPos values
VAR_IN_OUT
	CheckPos												:	VALUE_6D;
	Window													:	VALUE_6D;
END_VAR                 									
VAR CONSTANT            									
END_VAR
InPosAC													 	:= CAM(CheckPos.A, A ,Window.A)
																AND CAM(CheckPos.C, C ,Window.C);
END_METHOD

METHOD PUBLIC inPosByAxisNo : BOOL //Return value = TRUE selected axis is within window of checkPos values
VAR_INPUT
	No					:	INT;
END_VAR
VAR_IN_OUT
	CheckPos			:	VALUE_6D;
	Window				:	VALUE_6D;
END_VAR
inPosByAxisNo													:= (CAM(CheckPos.X, X ,Window.X) OR No <> 1)
																AND (CAM(CheckPos.Y, Y ,Window.Y) OR No <> 2)
																AND (CAM(CheckPos.Z, Z ,Window.Z) OR No <> 3)
																AND (CAM(CheckPos.A, A ,Window.A) OR No <> 4)
																AND (CAM(CheckPos.B, B ,Window.B) OR No <> 5)
																AND (CAM(CheckPos.C, C ,Window.C) OR No <> 6);
END_METHOD

METHOD PUBLIC inPosXY : BOOL //Return value = TRUE if axes are within window of checkPos values
VAR_IN_OUT
	CheckPos												:	VALUE_6D;
	Window													:	VALUE_6D;
END_VAR                 									
VAR CONSTANT            									
END_VAR
InPosXY													 	:= CAM(CheckPos.X, X ,Window.X)
																AND CAM(CheckPos.Y, Y ,Window.Y);
END_METHOD

METHOD PUBLIC InPosXYZ : BOOL //Return value = TRUE if axes are within window of checkPos values
VAR_IN_OUT
	CheckPos												:	VALUE_6D;
	Window													:	VALUE_6D;
END_VAR                 									
VAR CONSTANT            									
END_VAR
InPosXYZ												 	:= CAM(CheckPos.X, X ,Window.X)
																AND CAM(CheckPos.Y, Y ,Window.Y)
																AND CAM(CheckPos.Z, Z ,Window.Z);
END_METHOD

METHOD PUBLIC inPosXZ : BOOL //Return value = TRUE if axes are within window of checkPos values
VAR_IN_OUT
	CheckPos												:	VALUE_6D;
	Window													:	VALUE_6D;
END_VAR                 									
VAR CONSTANT            									
END_VAR
InPosXZ												 	:= CAM(CheckPos.X, X ,Window.X)
																AND CAM(CheckPos.Z, Z ,Window.Z);
END_METHOD

METHOD PUBLIC inPosYZ : BOOL //Return value = TRUE if axes are within window of checkPos values
VAR_IN_OUT
	CheckPos												:	VALUE_6D;
	Window													:	VALUE_6D;
END_VAR                 									
VAR CONSTANT            									
END_VAR
InPosYZ													 	:= CAM(CheckPos.Y, Y ,Window.Y)
																AND CAM(CheckPos.Z, Z ,Window.Z);
END_METHOD

METHOD PUBLIC reset : BOOL //Delete data and reset valid , TRUE if execution finished
VAR_INPUT
END_VAR
Delete(); 
Valid														:= FALSE;
reset														:= TRUE;
END_METHOD

END_FUNCTION_BLOCK

// POUs/Safety/Diag/SafetyIODeviceDiag_wEvents
{attribute 'no_check'}
FUNCTION_BLOCK SafetyIODeviceDiag_wEvents
VAR CONSTANT
	MIN_EVENT												:	INT := 1;
	MAX_EVENT												:	INT := 10;
	
//Event conn diag code xxxx					| FB1 - Msg 1..15
//Event conn diag code .4 					| FB2 - Msg 16
//Event conn diag code .5 					| FB3 - Msg 17
                                        	
//Event internal error 						| FB1 - Msg 18
                                        	
//Event send TextId 						| FB4 - Msg 19
                                        	
//Event send AX5xxx Err Chn 1 				| FB5 - Msg 20
//Event send AX5xxx Err Chn 1 				| FB6 - Msg 21
                                        	
//Event send Ex19 Err Debug 0x800E:0A 		| FB4 - Msg 22
//Event send Ex19 Err Debug 0x800E:0B		| FB5 - Msg 23
//Event send Ex19 Err Debug 0x800E:0C 		| FB6 - Msg 24
//Event send Ex19 Err Debug 0x800E:0D 		| FB7 - Msg 25
//Event send Ex19 Err Debug 0x800E:13 		| FB8 - Msg 26
//Event send Ex19 Err Debug 0x800E:14 		| FB9 - Msg 27
//Event send Ex19 Err Debug 0x800E:15		| FB10- Msg 28
                                        	
//Event send EL29 Err Debug 0x800E:0C 		| FB4 - Msg 30 (Querschluss bit 0..3)
//Event send EL29 Err Debug 0x800E:0C 		| FB4 - Msg 31 (Open load bit 4..7)
//Event send EL29 Err Debug 0x800E:0D		| FB5 - Msg 32
//Event send EL29 Err Debug 0x800E:0E 		| FB6 - Msg 33
//Event send EL29 Err Debug 0x800E:0E 		| FB7 - Msg 34
//Event send EL29 Err Debug 0x800E:0E 		| FB8 - Msg 35

                                        	
//Event send EK19 Err Debug 0x800E:0A		| FB4 - Msg 22 
//Event send EK19 Err Debug 0x800E:0B		| FB5 - Msg 23 
//Event send EK19 Err Debug 0x800E:0C 		| FB6 - Msg 24 
//Event send EK19 Err Debug 0x800E:0D 		| FB7 - Msg 25 
//Event send EK19 Err Debug 0x800E:0E	 	| FB8 - Msg 36..45
END_VAR
VAR_INPUT
	Enable													:	BOOL;	//FB will be processed as long as enable is TRUE 
	ConfirmTrig												:	BOOL;	//Resets error with rising edge 
	SourceId												:	UDINT;	//Multisource id 
	EcMasterDevId											:	UINT;	//Map to EtherCAT Master DevId
END_VAR                 									
VAR_OUTPUT              									
	Connected												:	BOOL;
	{attribute 'displaymode':='binary'}
	Status													:	DWORD;	//current status of event
	NoOfActiveEvents										:	INT;
END_VAR                 									

VAR(* internal *)
	state													:	INT := 0;
	{attribute 'displaymode':='binary'}
	ConnMsgDiagCode											:	BYTE;
	Read													:	SafetyIODeviceDiagRead;
   	Event													:	ARRAY [MIN_EVENT..MAX_EVENT] OF EventHandling; 
	DevTypeAndAddr											:	STRING(30);
    DebugData												:	 word;                 								                            	
	i														:	INT;
END_VAR

(* Safety IO device diag with events		V2	*)
(************************************************)

(* Status connected ***************************************************)
	Connected 												:= Read.AdsAddr.port <> 0;
	
(* Read adress and type ***********************************************)
	IF Enable AND Connected AND Read.MsgInfoDiag <> 0 OR State <> 0
	THEN
		CASE State OF
		0:	
			IF Read.MsgInfoDiag <> 0
			THEN
				Read(Execute := FALSE);
				Read(Execute := TRUE, EcMasterDevId := EcMasterDevId);
				State										:= State + 1;
			END_IF
			
		1: //Read diag data from device
			Read(Execute := TRUE, EcMasterDevId := EcMasterDevId);
			IF NOT Read.Busy
			THEN
	
				IF Read.Error
				THEN
					Event[1].Text1							:= SEL(Read.Name = '',Read.Name , '<ERR_READ_DIAG>');
					DevTypeAndAddr							:= SEL(Read.DevType = '', Read.DevType, '<Unknown>');
					DevTypeAndAddr							:= CONCAT(DevTypeAndAddr, CONCAT(' (Ec Addr.', CONCAT(TO_STRING(Read.AdsAddr.port),')')));	
					Event[1].Text2							:= CONCAT(' - ErrorID ', DWORD_TO_HEXSTR(TO_DWORD(Read.ErrorID),4,FALSE));
					Event[1].Text2							:= CONCAT(Event[1].Text2 , CONCAT(' in state ', TO_STRING(Read.DiagMsgTextId)));
					Event[1].SourceId						:= SourceId;
					Event[1].Flag							:= TRUE;
					State									:= 98;
				ELSIF Event[1].SourceId = 0
				THEN //Init device information 
					FOR i := MIN_EVENT TO MAX_EVENT
					DO
						Event[i].Text1						:= Read.Name;
						DevTypeAndAddr						:= CONCAT(Read.DevType, ' (FSOE Addr.');
						DevTypeAndAddr						:= CONCAT(DevTypeAndAddr, CONCAT(TO_STRING(Read.FSOEAddr), ')'));	
						Event[i].SourceId					:= SourceId;
					END_FOR
					State									:= 99;
				ELSE
					State									:= 99;
				END_IF		
				Read(Execute := FALSE);
			END_IF
			
		98: //Show internal error
			Event[1](
				Flag	:= Event[1].Flag AND NOT Event[1].ConfirmTrig,
				ConfirmTrig:= ConfirmTrig OR Read.MsgInfoDiag = 0, 
				MsgId	:= 18, 
				pText3	:= ADR(DevTypeAndAddr),
				Status	=> Status);	
			IF NOT Event[1].Status.31 
			THEN
				NoOfActiveEvents							:= 0;
				state										:= 0;
			ELSE
				NoOfActiveEvents							:= 1;
			END_IF
			
		99: //Fire events
			IF Read.MsgInfoDiag = 0 AND NOT Status.31
			THEN //Go back to 0 if messages cleared
				State 										:= 0;
			ELSE
				//Show connection error events
				_eventsConnDiag();
				
				//Fire device events
				IF Read.pDebugData <> 0 
				THEN //Safety devices without diag history object
					IF Read.DebugDataMaxId = 16#08 AND_THEN FIND(Read.DevType, 'AX580') <> 0
					THEN
						_eventsAX580x(Read.MsgInfoDiag <> 0);
					ELSIF Read.DebugDataMaxId = 16#10 AND_THEN Read.DevType = 'EL2904'
					THEN
						_eventsEL2904(Read.MsgInfoDiag <> 0);
					ELSIF Read.DebugDataMaxId = 16#40 AND_THEN Read.DevType = 'EK1914' 
					THEN
						_eventsEK1914(Read.MsgInfoDiag <> 0);
					ELSIF Read.DebugDataMaxId >= 16#10 
					THEN//EL1904 or EP1908
						_eventsEx190x(Read.MsgInfoDiag <> 0);		
					ELSE //Show internal error 
						Event[4](
							Flag	:= Read.MsgInfoDiag <> 0,
							ConfirmTrig:= ConfirmTrig OR Read.MsgInfoDiag = 0, 
							MsgId	:= 18, 
							Text2	:= CONCAT(' Invalid lenght of Coe object 0x800E for device ', TO_STRING(Read.DebugDataMaxId)),
							pText3	:= ADR(DevTypeAndAddr));	
					END_IF
				ELSE //TwinSAFE terminal with diag history  
					_eventsDiagHistory(Read.MsgInfoDiag <> 0);
				END_IF			
			END_IF		
						   	
			//Check whether one event is active **************************************
			NoOfActiveEvents 		 						:= 0;			
			Status											:= 0;						
			FOR i := MIN_EVENT TO MAX_EVENT
			DO 
				IF Event[i].Status.31 THEN NoOfActiveEvents := NoOfActiveEvents + 1 ; END_IF
				Status										:= Status OR Event[i].Status;
			END_FOR
		END_CASE
	END_IF

(*******************************************************************************)

METHOD PRIVATE _eventsAX580x : BOOL
VAR_INPUT
	ShowEvent										:	BOOL;
END_VAR
(* Fire AX5000 events ***********************************)
	//Send AX58xx diag code channel 1 
	IF Read.pDebugData^[1] = 0
	THEN
		Event[5].Text2										:= CONCAT('0x',DWORD_TO_HEXSTR(TO_DWORD(Read.pDebugData^[7]),4,FALSE));
	ELSE
		Event[5].Text2										:= '<Set CoE object 0xFA10:01 = 0>';
	END_IF
 
	Event[5](
		Flag	:= ShowEvent AND Read.msgSevyIsError ,
		ConfirmTrig:= ConfirmTrig, 
		MsgId	:= 20, 
		eClass	:= ,
		pText3	:= ADR(DevTypeAndAddr));	
		
	//Send AX58xx diag code channel 2
	IF Read.pDebugData^[1] = 0
	THEN
		Event[6].Text2										:= CONCAT('0x',DWORD_TO_HEXSTR(TO_DWORD(Read.pDebugData^[8]),4,FALSE));
	ELSE
		Event[6].Text2										:=  '<Set CoE object 0xFA10:01 = 0>';
	END_IF
 
	Event[6](
		Flag	:= ShowEvent AND Read.msgSevyIsError ,
		ConfirmTrig:= ConfirmTrig, 
		MsgId	:= 21, 
		eClass	:= ,
		pText3	:= ADR(Read.Name));

(******************************************************)
END_METHOD

METHOD PRIVATE _eventsConnDiag : BOOL
VAR_INPUT
END_VAR
(* Fire event for connection error code ************************************)
	ConnMsgDiagCode											:= 16#0F AND Read.MsgInfoDiag; 
	IF ConnMsgDiagCode <> 0 OR Event[1].Status.31
	THEN
		Event[1](
			Flag	:= ConnMsgDiagCode <> 0 AND NOT (ConnMsgDiagCode = 2#1101 AND Read.MsgInfoDiag.5),
			ConfirmTrig:= ConfirmTrig, 
			MsgId	:= ConnMsgDiagCode,  //1..15 		
			pText3	:= ADR(DevTypeAndAddr));	
	END_IF
	
	//Fire event xxx1 xxxx FSoE Slave error detected
	IF Read.MsgInfoDiag.4 OR Event[2].Status.31
	THEN
		Event[2](
			Flag	:= Read.MsgInfoDiag.4,
			ConfirmTrig:= ConfirmTrig, 
			MsgId	:= 16,		
			pText3	:= ADR(DevTypeAndAddr));	
	END_IF

(*
	//Fire event xx1x xxxx FSoE Slave notifies Failsafe Value active
	IF Read.MsgInfoDiag.5 OR Event[3].Status.31
	THEN
		Event[3](
			Flag	:= Read.MsgInfoDiag.5,
			ConfirmTrig:= ConfirmTrig, 
			MsgId	:= 17,		
			pText3	:= ADR(DevTypeAndAddr));		
	END_IF
*)	
	(*
	Tabelle 2-4: Diagnose-Informationen einer Connection
	Wert Beschreibung
	xxxx 0001 invalid command
	xxxx 0010 unknown command
	xxxx 0011 invalid connection ID
	xxxx 0100 invalid CRC
	xxxx 0101 Watchdog run out of time
	xxxx 0110 invalid FSoE-Adress
	xxxx 0111 invalid data
	xxxx 1000 invalid length of communicatoin parameter Kommunikationsparameterlänge
	xxxx 1001 invalid communicatoin parameter
	xxxx 1010 invalid operator parameter length
	xxxx 1011 invalid operator parameter
	xxxx 1100 FSoE Master Reset
	xxxx 1101 Module fault on slave detected with activated option "Modulfault is ComError"
	xxxx 1110 Module fault on EL290x at activated with option "Error achnowledge active"
	xxxx 1111 Slave not started or unexpected error argument
	
	*)
		
(***********************************************************************)
END_METHOD

METHOD PRIVATE _eventsDiagHistory : BOOL
VAR_INPUT
	ShowEvent										:	BOOL;
END_VAR
(* Send diag message textId ********************************************)
	Event[4](
		Flag	:= ShowEvent AND Read.msgSevyIsError ,
		ConfirmTrig:= ConfirmTrig, 
		MsgId	:= 19, 
		Text2	:= CONCAT('0x',DWORD_TO_HEXSTR(TO_DWORD(Read.DiagMsgTextId),4,FALSE)),
		pText3	:= ADR(DevTypeAndAddr));

(******************************************************)
END_METHOD

METHOD PRIVATE _eventsEK1914 : BOOL
VAR_INPUT
	ShowEvent										:	BOOL;
END_VAR
// Fire events for of EK1914 ****************************************)

		(* error during sensor-test *)
		Event[4].Flag 										:= Read.pDebugData^[16#0A] <> 0;
		IF Event[4].Flag OR Event[4].Status.31
		THEN
			DebugData										:= Read.pDebugData^[16#0A];
			Event[4].Text2									:= '';
			IF DebugData.0 THEN Event[4].Text2 				:= CONCAT(Event[4].Text2, '|1'); END_IF
			IF DebugData.1 THEN Event[4].Text2 				:= CONCAT(Event[4].Text2, '|2'); END_IF
		(*	IF DebugData.2 THEN Event[4].Text2 				:= CONCAT(Event[4].Text2, '|3'); END_IF
			IF DebugData.3 THEN Event[4].Text2 				:= CONCAT(Event[4].Text2, '|4');  END_IF
			IF DebugData.4 THEN Event[4].Text2 				:= CONCAT(Event[4].Text2, '|5'); END_IF
			IF DebugData.5 THEN Event[4].Text2 				:= CONCAT(Event[4].Text2, '|6'); END_IF
			IF DebugData.6 THEN Event[4].Text2 				:= CONCAT(Event[4].Text2, '|7'); END_IF
			IF DebugData.7 THEN Event[4].Text2 				:= CONCAT(Event[4].Text2, '|8');  END_IF *)
			Event[4].Text2 									:= CONCAT(Event[4].Text2, '|'); 			
			
			Event[4](
				Flag	:= ShowEvent ,
				ConfirmTrig:= ConfirmTrig, 
				MsgId	:= 22, 
				pText3	:= ADR(DevTypeAndAddr))	;
		END_IF

		(* Zweikanalauswertung fehlerhaft *)
		Event[5].Flag 										:= Read.pDebugData^[16#0B] <> 0;
		IF Event[5].Flag OR Event[5].Status.31
		THEN
			DebugData										:= Read.pDebugData^[16#0B];
			Event[5].Text2									:= '';
			IF DebugData.0 THEN Event[5].Text2 				:= CONCAT(Event[5].Text2, '|1+2'); END_IF
		(*	IF DebugData.1 THEN Event[5].Text2 				:= CONCAT(Event[5].Text2, '|3+4'); END_IF
			IF DebugData.2 THEN Event[5].Text2 				:= CONCAT(Event[5].Text2, '|5+6'); END_IF
			IF DebugData.3 THEN Event[5].Text2 				:= CONCAT(Event[5].Text2, '|7+8');  END_IF *)
			Event[5].Text2 									:= CONCAT(Event[5].Text2, '|'); 
			
			Event[5](
				Flag	:= ShowEvent ,
				ConfirmTrig:= ConfirmTrig, 
				MsgId	:= 23, 
				pText3	:= ADR(DevTypeAndAddr))	;
		END_IF

		(* Fehler Eingangspaar Trittmattenbetriebsart - Eingangspaar uneinig *)
		Event[6].Flag 										:= Read.pDebugData^[16#0C] <> 0;
		IF Event[6].Flag OR Event[6].Status.31
		THEN
			DebugData										:= Read.pDebugData^[16#0C];
			Event[6].Text2									:= '';
			IF DebugData.0 THEN Event[6].Text2 				:= CONCAT(Event[6].Text2, '|1+2'); END_IF
		(*	IF DebugData.1 THEN Event[6].Text2 				:= CONCAT(Event[6].Text2, '|3+4'); END_IF
			IF DebugData.2 THEN Event[6].Text2 				:= CONCAT(Event[6].Text2, '|5+6'); END_IF
			IF DebugData.3 THEN Event[6].Text2 				:= CONCAT(Event[6].Text2, '|7+8');  END_IF *)
			Event[6].Text2 									:= CONCAT(Event[6].Text2, '|'); 
			
			Event[6](
				Flag	:= ShowEvent ,
				ConfirmTrig:= ConfirmTrig, 
				MsgId	:= 24, 
				pText3	:= ADR(DevTypeAndAddr))	;
		END_IF

		(* Fehler Trittmattenbetriebsart Fremdeinspeisung *)
		Event[7].Flag 										:= Read.pDebugData^[16#0D] <> 0;
		IF Event[7].Flag OR Event[7].Status.31
		THEN
			DebugData										:= Read.pDebugData^[16#0D];
			Event[7].Text2									:= '';
			IF DebugData.0 THEN Event[7].Text2 				:= CONCAT(Event[7].Text2, '|1'); END_IF
			IF DebugData.1 THEN Event[7].Text2 				:= CONCAT(Event[7].Text2, '|2'); END_IF
		(*	IF DebugData.2 THEN Event[7].Text2 				:= CONCAT(Event[7].Text2, '|3'); END_IF
			IF DebugData.3 THEN Event[7].Text2 				:= CONCAT(Event[7].Text2, '|4');  END_IF
			IF DebugData.4 THEN Event[7].Text2 				:= CONCAT(Event[7].Text2, '|5'); END_IF
			IF DebugData.5 THEN Event[7].Text2 				:= CONCAT(Event[7].Text2, '|6'); END_IF
			IF DebugData.6 THEN Event[7].Text2 				:= CONCAT(Event[7].Text2, '|7'); END_IF
			IF DebugData.7 THEN Event[7].Text2 				:= CONCAT(Event[7].Text2, '|8');  END_IF *)
			Event[7].Text2 									:= CONCAT(Event[7].Text2, '|'); 
			
			Event[7](
				Flag	:= ShowEvent ,
				ConfirmTrig:= ConfirmTrig, 
				MsgId	:= 25, 
				pText3	:= ADR(DevTypeAndAddr))	;
		END_IF
		
		(* Fehler Ausgänge *)
		IF Read.pDebugData^[16#0E] <> 0 OR Event[8].Status.31 
		THEN
			DebugData										:= Read.pDebugData^[16#0E];
			
			CASE DebugData OF
			5:		Event[8].MsgId							:= 36;
			6:		Event[8].MsgId							:= 37;
			10:		Event[8].MsgId							:= 38;
			11:		Event[8].MsgId							:= 39;
			21..27:	Event[8].MsgId							:= 40;
			30..33:	Event[8].MsgId							:= 41;
			101:	Event[8].MsgId							:= 42;
			102:	Event[8].MsgId							:= 43;
			103:	Event[8].MsgId							:= 44;
			104:	Event[8].MsgId							:= 45;
			ELSE
				Event[8].MsgId								:= 0;
			END_CASE
				
			Event[8](
				Flag	:= ShowEvent AND Event[8].MsgId <> 0 ,
				ConfirmTrig:= ConfirmTrig, 
				MsgId	:= , 
				pText3	:= ADR(DevTypeAndAddr))	;
				
		END_IF		
(********************************************************************************)
END_METHOD

METHOD PRIVATE _eventsEL2904 : BOOL
VAR_INPUT
	ShowEvent										:	BOOL;
END_VAR
// Fire events for EL2904

	(* Fremeinspeisung oder Querschluss *)
	Event[4].Flag 										:= (Read.pDebugData^[16#0C] AND 16#000F) <> 0;
	IF Event[4].Flag OR Event[4].Status.31
	THEN
		DebugData										:= Read.pDebugData^[16#0C];
		Event[4].Text2									:= '';
		IF DebugData.0 THEN Event[4].Text2 				:= CONCAT(Event[4].Text2, '|1'); END_IF
		IF DebugData.1 THEN Event[4].Text2 				:= CONCAT(Event[4].Text2, '|2'); END_IF
		IF DebugData.2 THEN Event[4].Text2 				:= CONCAT(Event[4].Text2, '|3'); END_IF
		IF DebugData.3 THEN Event[4].Text2 				:= CONCAT(Event[4].Text2, '|4');  END_IF
		Event[4].Text2 									:= CONCAT(Event[4].Text2, '|'); 
			
		Event[4](
			Flag	:= ShowEvent ,
			ConfirmTrig:= ConfirmTrig, 
			MsgId	:= 30, 
			pText3	:= ADR(DevTypeAndAddr))	;
	END_IF

	(* Open load oder Mindeststrom (20mA) unterschritten, oder Maximalstrom ueberschritten (500mA) *)
	Event[5].Flag 										:= (Read.pDebugData^[16#0C] AND 16#00F0) <> 0;
	IF Event[5].Flag OR Event[5].Status.31
	THEN
		DebugData										:= Read.pDebugData^[16#0C];
		Event[5].Text2									:= '';
		IF DebugData.4 THEN Event[5].Text2 				:= CONCAT(Event[5].Text2, '|1'); END_IF
		IF DebugData.5 THEN Event[5].Text2 				:= CONCAT(Event[5].Text2, '|2'); END_IF
		IF DebugData.6 THEN Event[5].Text2 				:= CONCAT(Event[5].Text2, '|3'); END_IF
		IF DebugData.7 THEN Event[5].Text2 				:= CONCAT(Event[5].Text2, '|4');  END_IF
		Event[5].Text2 									:= CONCAT(Event[5].Text2, '|'); 
		
		Event[5](
			Flag	:= ShowEvent ,
			ConfirmTrig:= ConfirmTrig, 
			MsgId	:= 31, 
			pText3	:= ADR(DevTypeAndAddr));	
	END_IF
	
	(* Fehler Feldspannung Power Kontakte *)
	Event[6].Flag 										:= Read.pDebugData^[16#0D] <> 0;
	IF Event[6].Flag OR Event[6].Status.31
	THEN
		DebugData										:= Read.pDebugData^[16#0D];
		Event[6].Text2									:= '';
		IF DebugData.0 THEN 
			Event[6].Text2 								:= CONCAT(Event[6].Text2, '|Y'); 
		ELSE                                                                       
			Event[6].Text2 								:= CONCAT(Event[6].Text2, '|N'); 
		END_IF                                                                     
		IF DebugData.1 THEN                                                        
			Event[6].Text2 								:= CONCAT(Event[6].Text2, '|Y'); 
		ELSE                                                                       
			Event[6].Text2 								:= CONCAT(Event[6].Text2, '|N'); 
		END_IF
		Event[6].Text2 									:= CONCAT(Event[6].Text2, '|'); 
		
		Event[6](
			Flag	:= ShowEvent ,
			ConfirmTrig:= ConfirmTrig, 
			MsgId	:= 32, 
			pText3	:= ADR(DevTypeAndAddr))	;
	END_IF
	
	(* Temperaturfehler *)
	IF Read.pDebugData^[16#0E] <> 0 OR Event[7].Status.31 OR Event[8].Status.31 OR Event[9].Status.31
	THEN
		DebugData										:= Read.pDebugData^[16#0E];
		
		//Uebertemperatur
		Event[7](
			Flag	:= ShowEvent AND(DebugData.0 OR DebugData.1 OR DebugData.2),
			ConfirmTrig:= ConfirmTrig, 
			MsgId	:= 33, 
			pText3	:= ADR(DevTypeAndAddr));	
			
		//Untertemperatur
		Event[8](
			Flag	:= ShowEvent AND(DebugData.3 OR DebugData.4 OR DebugData.5),
			ConfirmTrig:= ConfirmTrig, 
			MsgId	:= 34, 
			pText3	:= ADR(DevTypeAndAddr))	;
			
		//Temp. Differenz
		Event[9](
			Flag	:= ShowEvent AND(DebugData.6 OR DebugData.6),
			ConfirmTrig:= ConfirmTrig, 
			MsgId	:= 35, 
			pText3	:= ADR(DevTypeAndAddr))	;
	END_IF
		
(***********************************************************************)
END_METHOD

METHOD PRIVATE _eventsEx190x : BOOL
VAR_INPUT
	ShowEvent										:	BOOL;
END_VAR
VAR
	DebugData												:	WORD;
END_VAR
// Fire events for EL1904 and EP1908 errors

	(* error during sensor-test *)
	Event[4].Flag 										:= Read.pDebugData^[16#0A] <> 0;
	IF Event[4].Flag OR Event[4].Status.31
	THEN
		DebugData										:= Read.pDebugData^[16#0A];
		Event[4].Text2									:= '';
		IF DebugData.0 THEN Event[4].Text2 				:= CONCAT(Event[4].Text2, '|1'); END_IF
		IF DebugData.1 THEN Event[4].Text2 				:= CONCAT(Event[4].Text2, '|2'); END_IF
		IF DebugData.2 THEN Event[4].Text2 				:= CONCAT(Event[4].Text2, '|3'); END_IF
		IF DebugData.3 THEN Event[4].Text2 				:= CONCAT(Event[4].Text2, '|4');  END_IF
		IF DebugData.4 THEN Event[4].Text2 				:= CONCAT(Event[4].Text2, '|5'); END_IF
		IF DebugData.5 THEN Event[4].Text2 				:= CONCAT(Event[4].Text2, '|6'); END_IF
		IF DebugData.6 THEN Event[4].Text2 				:= CONCAT(Event[4].Text2, '|7'); END_IF
		IF DebugData.7 THEN Event[4].Text2 				:= CONCAT(Event[4].Text2, '|8');  END_IF
		Event[4].Text2 									:= CONCAT(Event[4].Text2, '|'); 
		
		Event[4](
			Flag	:= ShowEvent ,
			ConfirmTrig:= ConfirmTrig, 
			MsgId	:= 22, 
			pText3	:= ADR(DevTypeAndAddr))	;
	END_IF

	(* Zweikanalauswertung fehlerhaft *)
	Event[5].Flag 										:= Read.pDebugData^[16#0B] <> 0;
	IF Event[5].Flag OR Event[5].Status.31
	THEN
		DebugData										:= Read.pDebugData^[16#0B];
		Event[5].Text2									:= '';
		IF DebugData.0 THEN Event[5].Text2 				:= CONCAT(Event[5].Text2, '|1+2'); END_IF
		IF DebugData.1 THEN Event[5].Text2 				:= CONCAT(Event[5].Text2, '|3+4'); END_IF
		IF DebugData.2 THEN Event[5].Text2 				:= CONCAT(Event[5].Text2, '|5+6'); END_IF
		IF DebugData.3 THEN Event[5].Text2 				:= CONCAT(Event[5].Text2, '|7+8');  END_IF
		Event[5].Text2 									:= CONCAT(Event[5].Text2, '|'); 		
	
		Event[5](
			Flag	:= ShowEvent ,
			ConfirmTrig:= ConfirmTrig, 
			MsgId	:= 23, 
			pText3	:= ADR(DevTypeAndAddr))	;
	END_IF

	(* Fehler Eingangspaar Trittmattenbetriebsart - Eingangspaar uneinig *)
	Event[6].Flag 										:= Read.pDebugData^[16#0C] <> 0;
	IF Event[6].Flag OR Event[6].Status.31
	THEN
		DebugData										:= Read.pDebugData^[16#0C];
		Event[6].Text2									:= '';
		IF DebugData.0 THEN Event[6].Text2 				:= CONCAT(Event[6].Text2, '|1+2'); END_IF
		IF DebugData.1 THEN Event[6].Text2 				:= CONCAT(Event[6].Text2, '|3+4'); END_IF
		IF DebugData.2 THEN Event[6].Text2 				:= CONCAT(Event[6].Text2, '|5+6'); END_IF
		IF DebugData.3 THEN Event[6].Text2 				:= CONCAT(Event[6].Text2, '|7+8');  END_IF
		Event[6].Text2 									:= CONCAT(Event[6].Text2, '|'); 
				
		Event[6](
			Flag	:= ShowEvent ,
			ConfirmTrig:= ConfirmTrig, 
			MsgId	:= 24, 
			pText3	:= ADR(DevTypeAndAddr))	;
	END_IF

	(* Fehler Trittmattenbetriebsart Fremdeinspeisung *)
	Event[7].Flag 										:= Read.pDebugData^[16#0D] <> 0;
	IF Event[7].Flag OR Event[7].Status.31
	THEN
		DebugData										:= Read.pDebugData^[16#0D];
		Event[7].Text2									:= '';
		IF DebugData.0 THEN Event[7].Text2 				:= CONCAT(Event[7].Text2, '|1'); END_IF
		IF DebugData.1 THEN Event[7].Text2 				:= CONCAT(Event[7].Text2, '|2'); END_IF
		IF DebugData.2 THEN Event[7].Text2 				:= CONCAT(Event[7].Text2, '|3'); END_IF
		IF DebugData.3 THEN Event[7].Text2 				:= CONCAT(Event[7].Text2, '|4');  END_IF
		IF DebugData.4 THEN Event[7].Text2 				:= CONCAT(Event[7].Text2, '|5'); END_IF
		IF DebugData.5 THEN Event[7].Text2 				:= CONCAT(Event[7].Text2, '|6'); END_IF
		IF DebugData.6 THEN Event[7].Text2 				:= CONCAT(Event[7].Text2, '|7'); END_IF
		IF DebugData.7 THEN Event[7].Text2 				:= CONCAT(Event[7].Text2, '|8');  END_IF
		Event[7].Text2 									:= CONCAT(Event[7].Text2, '|'); 
		
		Event[7](
			Flag	:= ShowEvent ,
			ConfirmTrig:= ConfirmTrig, 
			MsgId	:= 25, 
			pText3	:= ADR(DevTypeAndAddr))	;
	END_IF
	

//Events for EP1908 ****************************************************************)
IF Read.DebugDataMaxId > 16#10 THEN

	(* Fehler der Drehzahlueberwachung:Ueberdrehzahl *)
	Event[8].Flag 										:= Read.pDebugData^[16#13] <> 0;
	IF Event[8].Flag OR Event[8].Status.31
	THEN
		DebugData										:= Read.pDebugData^[16#13];
		Event[8].Text2									:= '';
		IF DebugData.0 THEN Event[8].Text2 				:= CONCAT(Event[8].Text2, '|1'); END_IF
		IF DebugData.1 THEN Event[8].Text2 				:= CONCAT(Event[8].Text2, '|2'); END_IF
		IF DebugData.2 THEN Event[8].Text2 				:= CONCAT(Event[8].Text2, '|3'); END_IF
		IF DebugData.3 THEN Event[8].Text2 				:= CONCAT(Event[8].Text2, '|4');  END_IF
		IF DebugData.4 THEN Event[8].Text2 				:= CONCAT(Event[8].Text2, '|5'); END_IF
		IF DebugData.5 THEN Event[8].Text2 				:= CONCAT(Event[8].Text2, '|6'); END_IF
		IF DebugData.6 THEN Event[8].Text2 				:= CONCAT(Event[8].Text2, '|7'); END_IF
		IF DebugData.7 THEN Event[8].Text2 				:= CONCAT(Event[8].Text2, '|8');  END_IF
		Event[8].Text2 									:= CONCAT(Event[8].Text2, '|'); 
		
		Event[8](
			Flag	:= ShowEvent ,
			ConfirmTrig:= ConfirmTrig, 
			MsgId	:= 26, 
			pText3	:= ADR(DevTypeAndAddr))	;
	END_IF
	
	(* Fehler in der Betriebsart: Two Channel Sync Velocity *)
	Event[9].Flag 										:= Read.pDebugData^[16#14] <> 0;
	IF Event[9].Flag OR Event[9].Status.31
	THEN
		DebugData										:= Read.pDebugData^[16#14];
		Event[9].Text2									:= '';
		IF DebugData.0 THEN Event[9].Text2 				:= CONCAT(Event[9].Text2, '|1+2'); END_IF
		IF DebugData.1 THEN Event[9].Text2 				:= CONCAT(Event[9].Text2, '|3+4'); END_IF
		IF DebugData.2 THEN Event[9].Text2 				:= CONCAT(Event[9].Text2, '|5+6'); END_IF
		IF DebugData.3 THEN Event[9].Text2 				:= CONCAT(Event[9].Text2, '|7+8');  END_IF
		Event[9].Text2 									:= CONCAT(Event[9].Text2, '|'); 
		
		Event[9](
			Flag	:= ShowEvent ,
			ConfirmTrig:= ConfirmTrig, 
			MsgId	:= 27, 
			pText3	:= ADR(DevTypeAndAddr))	;
	END_IF
	
	(* Fehler in der Betriebsart: Two Channel Sync Velocity UND Two Channel Encoder Velocity Control*)
	Event[10].Flag 										:= Read.pDebugData^[16#15] <> 0;
	IF Event[10].Flag OR Event[10].Status.31
	THEN
		DebugData										:= Read.pDebugData^[16#15];
		Event[10].Text2									:= '';
		IF DebugData.0 THEN Event[10].Text2 			:= CONCAT(Event[10].Text2, '|1+2'); END_IF
		IF DebugData.1 THEN Event[10].Text2 			:= CONCAT(Event[10].Text2, '|3+4'); END_IF
		IF DebugData.2 THEN Event[10].Text2 			:= CONCAT(Event[10].Text2, '|5+6'); END_IF
		IF DebugData.3 THEN Event[10].Text2 			:= CONCAT(Event[10].Text2, '|7+8');  END_IF
		Event[10].Text2 								:= CONCAT(Event[10].Text2, '|'); 
		
		Event[10](
			Flag	:= ShowEvent ,
			ConfirmTrig:= ConfirmTrig, 
			MsgId	:= 28, 
			pText3	:= ADR(DevTypeAndAddr))	;
	END_IF
END_IF

(************************************************************************************)
END_METHOD

END_FUNCTION_BLOCK

// POUs/Safety/Diag/SafetyIODeviceDiagRead
{attribute 'no_check'}
{attribute 'enable_dynamic_creation'}
FUNCTION_BLOCK SafetyIODeviceDiagRead EXTENDS FbBase
VAR CONSTANT
	bitTwinSAFETerm											:	BYTE := 0; //Ex1918,ELx9xx, etc. (2nd generation of TwinSAFE devices with CoE Index 10F3 Diag History included)
	bitSafetyTerm											:	BYTE := 1; //EL1904,EL2904,EK1914,EP1908 (Diagnoses provided via CoE Index 0x800E FSOE Internal Data, Debug 1..x) 
 	bitAX58xx												:	BYTE := 2; //AX5805,AX5806 (Diag via CoE index 0xFA10)
END_VAR
VAR_INPUT
	EcMasterDevId											:	UINT;	//EtherCAT Master DevId
END_VAR                 									
VAR_OUTPUT              									 
	AdsAddr											AT %I*	:	AMSADDR; //Link to terminal/box/device AMS Net Addr.
	{attribute 'displaymode':='binary'}
	MsgInfoDiag										AT %I*	:	USINT; 	//Link to connection messagediag of EL69xx (Needs to be enabled for alias of device)
//	{attribute 'displaymode':='hexadecimal'}
//	MsgInfoState									AT %I*	:	USINT; 	//Link to connection message state of EL69xx (Needs to be enabled for alias of device)	
	DevType													:	STRING(15); //CoE index 1008 / e.g. EL1908, EP1957-0022, etc...
	Name													:	STRING(31);	//Device name as defined in system manager configuration								
	FSoEAddr												:	WORD; //CoE index 0xF980
	DiagMsgSeverity											:	UINT; //Info (0) Warning (1) or Error (2)
	{attribute 'displaymode':='hexadecimal'}
	DiagMsgTextId											: 	UINT; //CoE Index 10F3 newest diagnoses message TextID (xyzz -> X =Type | y = Source | zz = Message ID)
	{attribute 'displaymode':='hexadecimal'}
	pDebugData												:	POINTER TO ARRAY[0..64] OF WORD; //Pointer to CoE index 0x800E - FSOE Internal Data - Debug 1-x for diag of "Safety Terminals" (or CoE Index 0xFA10 for AX58xx)
	DebugDataMaxId											:	UINT; //Max index for pointer pDebugData to array of word (Debug 1..x) if 0 data are invalid		
END_VAR                 									

VAR(* internal *)    
	{attribute 'displaymode':='bin'}
	DevCategory												:	BYTE;
	IOF_GetBoxNameByAddr									:	IOF_GetBoxNameByAddr := (TMOUT	:= DEFAULT_ADS_TIMEOUT);
	EcCoEReadDiagMsg										:	EcCoEReadNewestDiagMsg ;              									
	EcCoESdoReadEx											:	FB_EcCoESdoReadEx := (tTimeout := DEFAULT_ADS_TIMEOUT);       
	i														:	INT;  								                            	
END_VAR
(*
Tabelle 2-4: Diagnose-Informationen einer Connection
Wert Beschreibung
xxxx 0001 invalid command
xxxx 0010 unknown command
xxxx 0011 invalid connection ID
xxxx 0100 invalid CRC
xxxx 0101 Watchdog run out of time
xxxx 0110 invalid FSoE-Adress
xxxx 0111 invalid data
xxxx 1000 invalid length of communicatoin parameter Kommunikationsparameterlänge
xxxx 1001 invalid communicatoin parameter
xxxx 1010 invalid operator parameter length
xxxx 1011 invalid operator parameter
xxxx 1100 FSoE Master Reset
xxxx 1101 Module fault on slave detected with activated option "Modulfault is ComError"
xxxx 1110 Module fault on EL290x at activated with option "Error achnowledge active"
xxxx 1111 Slave not started or unexpected error argument

xxx1 xxxx FSoE Slave error detected
xx1x xxxx FSoE Slave notifies Failsafe Value active
x1xx xxxx StartUp
1xxx xxxx FSoE Master notifies Failsafe Value active
*)

(* IO Safety Terminal Status Diag		V2.0	*)
(************************************************)

(* Trigger to read diag **********************************************)
	rtExecute(CLK := Execute);
	
(* Read adress and type ***********************************************)
	CASE state OF
	0:
		Busy 												:= FALSE;
		IF NOT Execute
		THEN
			Done											:= FALSE;
			Error											:= FALSE;
			ErrorId											:= 0;					
		END_IF
		
		IF rtExecute.Q
		THEN
			Busy 											:= TRUE;
			Done											:= FALSE;
			Error											:= FALSE;
			ErrorId											:= 0;
			DiagMsgTextId									:= 0;
			DiagMsgSeverity									:= 0;

			EcCoESdoReadEx(bExecute := FALSE, bCompleteAccess := FALSE);
			IOF_GetBoxNameByAddr(Start := FALSE);
			EcCoEReadDiagMsg(Execute := FALSE);
			
			IF DevCategory.bitTwinSAFETerm
			THEN
				state 										:= 10;	
			ELSIF DevCategory.bitSafetyTerm
			THEN
				state 										:= SEL(DebugDataMaxId = 0, 21, 20);
			ELSIF DevCategory.bitAX58xx				
			THEN 
				state 										:= 30;
				
			ELSE //Read more device information 
				state										:= state + 1;				
			END_IF
		
		END_IF

	1: (* read FSOE adress *)
		EcCoESdoReadEx(
			sNetId			:= F_CreateAmsNetId(nIds := AdsAddr.netId ),
			nSlaveAddr		:= AdsAddr.port,
			nSubIndex		:= 16#1,
			nIndex			:= 16#F980,
			pDstBuf			:= ADR(FSOEAddr),
			cbBufLen		:= SIZEOF(FSOEAddr),
			bExecute		:= TRUE,
			tTimeout		:=  (* Default *),
			bCompleteAccess	:= False,
			bBusy			=> ,
			bError			=> ,
			nErrId			=> );
			
		IF NOT EcCoESdoReadEx.bBusy
		THEN
			IF EcCoESdoReadEx.bError 
			THEN
				Busy 										:= FALSE;
				Error										:= TRUE;
				ErrorId										:= EcCoESdoReadEx.nErrId;
				DiagMsgTextId								:= TO_UINT(state);
				state										:= 0;
			ELSE      									
				state 										:= state + 1;
			END_IF
			EcCoESdoReadEx(bExecute := FALSE);
		END_IF

	2: //Ready name from system manager configuration
		IOF_GetBoxNameByAddr(
			NETID		:='' , (* Local *)
			DEVICEID	:= UINT_TO_UDINT(EcMasterDevId) ,
			BOXADDR		:= AdsAddr.port ,
			START		:= EcMasterDevId <> 0,
			BOXNAME		=> );
			
		IF NOT IOF_GetBoxNameByAddr.Busy
		THEN
			IF IOF_GetBoxNameByAddr.Err 
			THEN
				Busy 										:= FALSE;
				Error										:= TRUE;
				ErrorId										:= IOF_GetBoxNameByAddr.ERRID;
				DiagMsgTextId								:= TO_UINT(state);
				state										:= 0;
			ELSIF IOF_GetBoxNameByAddr.Start
			THEN
				state 										:= state + 1;
			ELSE //No box name to read
				Name										:= CONCAT('EtherCAT Addr.',TO_STRING(AdsAddr.port));
			END_IF
			IOF_GetBoxNameByAddr(START := FALSE);
		END_IF
		
	3:  (* read device name e.g. EL1904 *)
		EcCoESdoReadEx(bExecute	:= TRUE, nIndex	:= 16#1008, nSubIndex := 16#0, pDstBuf := ADR(DevType),cbBufLen	:= SIZEOF(DevType), bCompleteAccess := FALSE);

		IF NOT EcCoESdoReadEx.bBusy
		THEN
			IF EcCoESdoReadEx.bError 
			THEN
				Busy 										:= FALSE;
				Error										:= TRUE;
				ErrorId										:= EcCoESdoReadEx.nErrId;
				DiagMsgTextId								:= TO_UINT(state);
				state										:= 0;
			ELSE       
				 //Delte type from name if in brakets 
				Name										:= DELETE(IOF_GetBoxNameByAddr.BOXNAME, LEN(DevType) + 2 , FIND(IOF_GetBoxNameByAddr.BOXNAME,DevType) - 1);
                             	
				IF DevType = 'AX5806' OR_ELSE DevType = 'AX5805'
				THEN
					DevCategory.bitAX58xx					:= TRUE;
					state 									:= 30;
				ELSIF DevType = 'EL1904' OR_ELSE DevType = 'EL2904' OR_ELSE DevType = 'EK1914' OR_ELSE DevType = 'EP1908'
				THEN
					DevCategory.bitSafetyTerm 				:= TRUE;
					state 									:= SEL(DebugDataMaxId = 0, 21, 20);
				ELSE
					DevCategory.bitTwinSAFETerm				:= TRUE;
					state 									:= 10;
				END_IF
				
			END_IF
			EcCoESdoReadEx(bExecute := FALSE);
		END_IF

	(* Read diagnoses latest entry from diag history ***********************************)	
	10: 
		EcCoEReadDiagMsg(Execute := TRUE, AdsAddr := AdsAddr);
		IF NOT EcCoEReadDiagMsg.Busy
		THEN
			IF EcCoEReadDiagMsg.Error 
			THEN
				Busy 										:= FALSE;
				Error										:= TRUE;
				ErrorId										:= EcCoEReadDiagMsg.ErrorID;
				DiagMsgTextId								:= TO_UINT(state);
				state										:= 0;				
			ELSE
				DiagMsgTextId								:= EcCoEReadDiagMsg.MsgId;
				DiagMsgSeverity								:= EcCoEReadDiagMsg.MsgSeverity;
				Done										:= TRUE;
				Busy										:= FALSE;
				State										:= 0;
			END_IF
		END_IF
		
	(* Read lenght of 0x800E:0 FSOE internal data.Debug terminal *********************************)
	20:
		EcCoESdoReadEx(bExecute	:= DebugDataMaxId = 0, nIndex	:= 16#800E, nSubIndex := 16#0, pDstBuf := ADR(DebugDataMaxId),cbBufLen	:= SIZEOF(DebugDataMaxId), bCompleteAccess := FALSE);

		IF NOT EcCoESdoReadEx.bBusy
		THEN
			IF EcCoESdoReadEx.bError 
			THEN
				Busy 										:= FALSE;
				Error										:= TRUE;
				ErrorId										:= EcCoESdoReadEx.nErrId;
				DiagMsgTextId								:= TO_UINT(state);
				state										:= 0;
			ELSIF DebugDataMaxId = 0
			THEN
				Busy 										:= FALSE;
				Error										:= TRUE;
				ErrorId										:= E_AdsErr.DEVICE_INVALIDPARM; //Lenght of index cannot be 0
				DiagMsgTextId								:= TO_UINT(state);
				state										:= 0;				
			ELSIF pDebugData = 0
			THEN                                  	
				pDebugData									:= __NEW(WORD,TO_UDINT(DebugDataMaxId + 1)); //e.g. 16 words = 32 bytes + 1 word for index 0 (which is in fact a byte  				
				IF PARAM.ENABLE_DEBUG_MSG_DYNAMIC_MEM_ALLOCATION
				THEN
					AdsLogHint('EngineeringToolbox | FB SafetyIOReadDiag | An instance allocated %s bytes from the dynamic memory of the ADS router memory pool', TO_STRING((DebugDataMaxId * 2) + 2));
				END_IF
				state 										:= state + 1;
			ELSE
				state 										:= state + 1;
			END_IF
			EcCoESdoReadEx(bExecute := FALSE);
		END_IF	
		
	21://Read all debug data from terminal
		EcCoESdoReadEx(bExecute	:= TRUE, nIndex	:= 16#800E, nSubIndex := 16#0, pDstBuf := pDebugData ,cbBufLen := TO_UDINT(DebugDataMaxId * 2) + SIZEOF(DebugDataMaxId) , bCompleteAccess := TRUE);

		IF NOT EcCoESdoReadEx.bBusy
		THEN
			IF EcCoESdoReadEx.bError 
			THEN
				IF pDebugData = 0
				THEN
					DebugDataMaxId							:= 0;
				END_IF
				Busy 										:= FALSE;
				Error										:= TRUE;
				ErrorId										:= EcCoESdoReadEx.nErrId;
				DiagMsgTextId								:= TO_UINT(state);
				state										:= 0;
			ELSE                                    		
				Done										:= TRUE;
				Busy										:= FALSE;
				DiagMsgSeverity								:= 2;
				State										:= 0;					
			END_IF
			EcCoESdoReadEx(bExecute := FALSE, bCompleteAccess := FALSE );
		END_IF			
	
	(* Read diag data from AX58xx *********************************)
	30:
		IF pDebugData = 0
		THEN
			DebugDataMaxId									:= 16#8;
			pDebugData										:= __NEW(WORD,TO_UDINT(DebugDataMaxId + 1));
			
			IF PARAM.ENABLE_DEBUG_MSG_DYNAMIC_MEM_ALLOCATION
			THEN
				AdsLogHint('EngineeringToolbox | FB SafetyIOReadDiag | An instance allocated %s bytes from the dynamic memory of the ADS router memory pool', '18');
			END_IF				
		END_IF
		
		EcCoESdoReadEx(bExecute	:= TRUE, nIndex	:= 16#FA10, nSubIndex := 16#0, pDstBuf := pDebugData, cbBufLen	:= TO_UDINT(DebugDataMaxId * 2) + SIZEOF(DebugDataMaxId),bCompleteAccess := TRUE);

		IF NOT EcCoESdoReadEx.bBusy
		THEN
			IF EcCoESdoReadEx.bError 
			THEN
				IF pDebugData = 0
				THEN
					DebugDataMaxId							:= 0;
				END_IF
				Busy 										:= FALSE;
				Error										:= TRUE;
				ErrorId										:= EcCoESdoReadEx.nErrId;
				DiagMsgTextId								:= TO_UINT(state);
				state										:= 0;
			ELSE                                    		
				Done										:= TRUE;
				Busy										:= FALSE;
				DiagMsgSeverity								:= 2;
				State										:= 0;	
			END_IF
			EcCoESdoReadEx(bExecute := FALSE, bCompleteAccess := FALSE);
		END_IF	
	ELSE
		;
	END_CASE
			
(*********************************************************************************************)

METHOD FB_exit : BOOL
VAR_INPUT
	bInCopyCode : BOOL; // if TRUE, the exit method is called for exiting an instance that is copied afterwards (online change).
END_VAR
IF NOT bInCopyCode AND pDebugData <> 0
THEN //Release memory in case the PLC stopps
	__DELETE(pDebugData);
	DebugDataMaxId								:= 0;
END_IF
END_METHOD

{attribute 'monitoring' := 'call'}
PROPERTY PUBLIC msgSevyIsError : BOOL
GET
msgSevyIsError := DiagMsgSeverity = 2;
END_GET
END_PROPERTY

{attribute 'monitoring' := 'call'}
PROPERTY PUBLIC msgSevyIsInfo : BOOL
GET
msgSevyIsInfo := DiagMsgSeverity = 0;
END_GET
END_PROPERTY

{attribute 'monitoring' := 'call'}
PROPERTY PUBLIC msgSevyIsWarning : BOOL
GET
msgSevyIsWarning := DiagMsgSeverity = 1;
END_GET
END_PROPERTY

END_FUNCTION_BLOCK

// POUs/Safety/Diag/SafetyIOsDiag
{attribute 'no_check'}
FUNCTION_BLOCK SafetyIOsDiag
VAR CONSTANT
	MIN_TERM												:	INT := 1;
	MAX_TERM												:	INT := PARAM.SAFETY_IO_TERM_DIAG_MAX;
END_VAR                     								
VAR_INPUT                   								
	Enable													:	BOOL;	//FB will be processed as long as enable is TRUE 
	ConfirmTrig												:	BOOL;	//Resets error with rising edge 
	SourceMultiId											:	UDINT := 100310;
	EcMasterDevId											:	UINT;	//Map to EtherCAT Master DevId
END_VAR                     								
VAR_OUTPUT                  	
	{attribute 'displaymode':='binary'}
	Status													:	DWORD;	//Current status of all events
	NoOfActiveEvents										:	INT;
END_VAR
VAR (* Events/Blocks/Var internal *)
	DevNo													:	ARRAY [MIN_TERM..MAX_TERM] OF SafetyIODeviceDiag_wEvents;
    tonStartupDelay											:	ton := (PT := T#200MS);                 								
	i														:	INT := MIN_TERM;
	StartCnt												:	BYTE := 0;
                           	
END_VAR

(* EL Safety IO Terminal Diag							*)
(********************************************************)

(* start one after the other ***************************)
	IF StartCnt < MAX_TERM 
	THEN
		tonStartupDelay(IN := TRUE);
		IF tonStartupDelay.Q
		THEN
			tonStartupDelay(IN := FALSE);
			StartCnt 										:= StartCnt + 1;
			DevNo[StartCnt].SourceId						:= SourceMultiId + StartCnt;
			DevNo[StartCnt].EcMasterDevId					:= EcMasterDevId;
			
		END_IF
	END_IF

(* terminal event ***************************************)
	Status 													:= 0;
	NoOfActiveEvents										:= 0;
	FOR i := MIN_TERM TO MAX_TERM
	DO
		DevNo[i](
			Enable			:= Enable AND StartCnt >= i,
			ConfirmTrig		:= ConfirmTrig,
			SourceId		:= ,
			EcMasterDevId	:= ,
			Status			=> );
				
		IF DevNo[i].Connected
		THEN
			IF DevNo[i].Status.31 THEN NoOfActiveEvents := NoOfActiveEvents + DevNo[i].NoOfActiveEvents ; END_IF
			Status											:= Status OR DevNo[i].Status;
		ELSE
			EXIT; 
		END_IF
	END_FOR

(*******************************************************)

END_FUNCTION_BLOCK

// POUs/Safety/Diag/SafetyLogicAndIOTerminalDiag
{attribute 'no_check'}
FUNCTION_BLOCK SafetyLogicAndIOTerminalDiag EXTENDS SafetyLogicTerminalDiag
VAR_OUTPUT CONSTANT
	MIN_IN_MODULE											:	INT := 1;
	MAX_IN_MODULE											:	INT := Param.SAFETY_LOGIC_IO_TERM_DIAG_MAX_MODULE; 
	MIN_OUT_MODULE											:	INT := 1;
	MAX_OUT_MODULE											:	INT := Param.SAFETY_LOGIC_IO_TERM_DIAG_MAX_MODULE; 	
END_VAR                 									
VAR_INPUT               									
	FSOUT_Module_Output								AT %Q*	:	ARRAY[MIN_OUT_MODULE..MAX_OUT_MODULE] OF BOOL;	
END_VAR
VAR_OUTPUT
	FSIN_Module_Fault								AT %I*	:	ARRAY[MIN_IN_MODULE..MAX_IN_MODULE] OF BOOL;
	FSOUT_Module_Fault								AT %I*	:	ARRAY[MIN_OUT_MODULE..MAX_OUT_MODULE] OF BOOL;

END_VAR
VAR 
END_VAR
VAR 
(* Events/Blocks/Var internal *)
	EventFSINModuleFault									:	EventHandling := (SourceId := DEFAULT_SOURCE_ID, MsgId:= 7);	
	EventFSOUTModuleFault									:	EventHandling := (SourceId := DEFAULT_SOURCE_ID, MsgId:= 8);
	
{attribute 'displaymode':='binary'}
	FSIN_Faults												:	DWORD; 
{attribute 'displaymode':='binary'}
	FSOUT_Faults											:	DWORD; 

END_VAR

(* Extension to ELx9xx Safety Logic with local IO's Terminal Diag	*)
(********************************************************************)

(* call super *************************************************************)
	SUPER^();
	
(* Event 7-8 *******************************************************************)
	FOR i := MIN_IN_MODULE TO MAX_IN_MODULE
	DO
		FSIN_Faults											:= CSETBIT32(FSIN_Faults,TO_SINT(i-1),FSIN_Module_Fault[i]);
	END_FOR
		
	EventFSINModuleFault(
		Flag		:= FSIN_Faults <> 0 AND_THEN IO.InfoDataState = Tc2_EtherCAT.EC_DEVICE_STATE_OP AND Enable,
		ConfirmTrig	:= Quit OR NOT Enable,
		MsgId		:= ,
		SourceId	:= ,
		eClass		:=,
		format		:= ,
		Text1		:= DWORD_TO_BINSTR_EXT(FSIN_Faults,MAX_IN_MODULE,3),
		Text2		:= ,
		pText3		:= ADR(IO.DevName),
		State		=> ,
		Status		=> );

	FOR i := MIN_OUT_MODULE TO MAX_OUT_MODULE
	DO
		FSOUT_Faults											:= CSETBIT32(FSOUT_Faults,TO_SINT(i-1),FSOUT_Module_Fault[i]);
	END_FOR
			 	
	EventFSOUTModuleFault(
		Flag		:= FSOUT_Faults <> 0 AND_THEN IO.InfoDataState = Tc2_EtherCAT.EC_DEVICE_STATE_OP AND Enable,
		ConfirmTrig	:= Quit OR NOT Enable,
		MsgId		:= ,
		SourceId	:= ,
		eClass		:=,
		format		:= ,
		Text1		:= DWORD_TO_BINSTR_EXT(FSIN_Faults,MAX_OUT_MODULE,3),
		Text2		:= ,
		pText3		:= ADR(IO.DevName),
		State		=> ,
		Status		=> );	
				
	Status													:= Status OR EventFSINModuleFault.Status OR EventFSOUTModuleFault.Status;
(*****************************************************************)

{attribute 'monitoring' := 'call'}
PROPERTY PUBLIC inputModuleFault : bool
GET
VAR
	i	: int;
END_VAR
inputModuleFault									:= FALSE;
FOR i := MIN_IN_MODULE TO MAX_IN_MODULE
DO
	IF FSIN_Module_Fault[i]
	THEN
		inputModuleFault							:= TRUE;
		EXIT;
	END_IF
	
END_FOR
END_GET
END_PROPERTY

{attribute 'monitoring' := 'call'}
PROPERTY PUBLIC moduleInFault : bool
GET
moduleInFault			:= inputModuleFault or outputModuleFault;
END_GET
END_PROPERTY

{attribute 'monitoring' := 'call'}
PROPERTY PUBLIC outputModuleFault : bool
GET
VAR
	i : int;
END_VAR
outputModuleFault									:= FALSE;
FOR i := MIN_OUT_MODULE TO MAX_OUT_MODULE
DO
	IF FSOUT_Module_Fault[i]
	THEN
		outputModuleFault							:= TRUE;
		EXIT;
	END_IF
	
END_FOR
END_GET
END_PROPERTY

END_FUNCTION_BLOCK

// POUs/StringHelper/DWORD_TO_BINSTR_EXT
{attribute 'no_check' := ''}
FUNCTION DWORD_TO_BINSTR_EXT : T_MaxString //This function converts a decimal number into a binary string (base 2), where the digits are separated according to the selected mode 
//e.g. 1111000011110000 -> 1111_0000_1111_0000 
VAR_INPUT
	In														: DWORD;//The decimal number requiring conversion.
	Precision												: INT; //Minimum number of displayed digits (digits), filled up with 0 from left if significant digits are less then that
	Mode													: INT; //1=Separate high and low word / 2=Separate bytes / 3=Separate nibbles /ELSE no separation | Separator = Param.DOWRD_TO_XXXSTR_EXT_SEPARATOR
END_VAR
VAR		
	k														:	INT;											
END_VAR

DWORD_TO_BINSTR_EXT 										:= DWORD_TO_BINSTR(in,precision);

CASE mode OF
1:// Separate by low word and high word
	DWORD_TO_BINSTR_EXT										:= INSERT_EXT(DWORD_TO_BINSTR_EXT, PARAM.XWORD_TO_XXXSTR_EXT_SEPARATOR ,16);
	
2://Separate by bytes
	DWORD_TO_BINSTR_EXT										:= INSERT_EXT(DWORD_TO_BINSTR_EXT,PARAM.XWORD_TO_XXXSTR_EXT_SEPARATOR,8);
	
3://Separate by nibble
	DWORD_TO_BINSTR_EXT										:= INSERT_EXT(DWORD_TO_BINSTR_EXT,PARAM.XWORD_TO_XXXSTR_EXT_SEPARATOR,4);
END_CASE

//Cut seperator at the end
k 															:= LEN(DWORD_TO_BINSTR_EXT);
IF k > 0 AND_THEN DWORD_TO_BINSTR_EXT[k-1] = PARAM.XWORD_TO_XXXSTR_EXT_SEPARATOR[0]
THEN
	DWORD_TO_BINSTR_EXT[k-1]								:= 0;
END_IF

END_FUNCTION

// POUs/StringHelper/INSERT_EXT
{attribute 'no_check' := ''}
FUNCTION INSERT_EXT : T_MaxString //The function INSERT_EXT inserts STR2 into STR1 at every ITERATION_POS position e.g. /r/n
VAR_INPUT
	STR1													:T_MaxString; //Base string - Hint! The base string will cut off if iteration of insertions exceeded the size of the string variable 
	STR2													:T_MaxString; //Insert string 
	ITERATION_POS											: INT; //Insert iteration position 
END_VAR
VAR
	Length1,length2,i,iEnd									: INT;														
END_VAR

INSERT_EXT													:= STR1;
Length1														:= LEN(STR1);
Length2														:= LEN(STR2);
IF TO_UINT(Length1 + Length2) > SIZEOF(STR1)
	OR ITERATION_POS = 0
THEN
	;
ELSE
	iEnd													:= MAX(1,ABS(Length1 / ITERATION_POS));
	FOR i := 1 TO iEnd
	DO 
		INSERT_EXT											:= INSERT(INSERT_EXT,STR2,(i*ITERATION_POS) + ((i-1)*Length2));
	END_FOR
END_IF

END_FUNCTION

// POUs/Safety/Diag/SafetyLogicTerminalDiag
{attribute 'no_check'}
FUNCTION_BLOCK SafetyLogicTerminalDiag // EL6910, EL and EP devices with integrated TwinSAFE logic 
VAR CONSTANT
	MIN_FB													:	INT := 1;
	MAX_FB													:	INT := PARAM.SAFETY_PLC_TERM_DIAG_MAX_FB;
	
	TIMEOUT_CYCLE_COUNTER									:	TIME := T#1S;
	DEFAULT_SOURCE_ID										:	UDINT := 100300; //Multisource id 
	INVALID_SAFETY_LOGIC_STATE								:	USINT := 255;
END_VAR                 									
VAR_INPUT               									
	Enable													:	BOOL := TRUE;	//FB will be processed as long as enable is TRUE 
	Quit													:	BOOL;			//Resets error with rising edge 
	IO														:	Eyx9xx;			
END_VAR
VAR_OUTPUT
	{attribute 'displaymode':='binary'}
	Status													:	DWORD; 			//current sttus of all events
	NoOfActiveEvents										:	INT;
END_VAR
VAR (* FunctionBlock Status *)
	FBInfoDataDiag	 								AT %I*	:	ARRAY [MIN_FB..MAX_FB] OF UINT; //Safety FB diagnostic information
END_VAR
VAR (* Events/Blocks/Var internal *)
//	EventInputSizeMism										: 	EventHandling := (MsgId:= 1); //Msg id 1 not used for logic terminals
//	EventOutputSizeMism										: 	EventHandling := (MsgId:= 2); //Msg id 1 not used for logic terminals
	EventInvalidCRC											:	EventHandling := (SourceId := DEFAULT_SOURCE_ID, MsgId:= 3);	
	EventCycleCounter										:	EventHandling := (SourceId := DEFAULT_SOURCE_ID, MsgId:= 4);
	EventLogicState											:	EventHandling := (SourceId := DEFAULT_SOURCE_ID, MsgId:= 5);
//	EventDiagHist											:	EventHandling := (SourceId := DEFAULT_SOURCE_ID, MsgId:= 6);
	
//	ReadDiagHist											:	SafetyIODeviceDiagRead;
		
	TON_CycleCounter										:	TON := (PT := TIMEOUT_CYCLE_COUNTER);
	MemCycleCounter											: 	USINT;
	
	EventFBError											:	ARRAY [MIN_FB..MAX_FB] OF EventHandling; //MsgId from 11 to MAX_FB + 10
                        									                        	
	i														:	INT := MIN_FB;

END_VAR

(* EL6910/ ELx9xx Safety Logic Terminal Diag	*)
(************************************************)

(* call IO *************************************************************)
	IO();
	
(* Event 3-10 *******************************************************************)
(* Events 1 and 2 only for EL6900 devices *)

	EventInvalidCRC(
		Flag		:= IO.ProjectCRC = 0 AND_THEN NOT IO.WcState AND IO.InfoDataState = Tc2_EtherCAT.EC_DEVICE_STATE_OP AND Enable,
		ConfirmTrig	:= Quit OR NOT Enable AND EventInvalidCRC.State <> TCEVENTSTATE_INVALID ,
		MsgId		:= ,
		SourceId	:= ,
		eClass		:=,
		format		:= ,
		Text1		:= ,
		Text2		:= ,
		pText3		:= ADR(IO.DevName),
		State		=> ,
		Status		=> );
			
	TON_CycleCounter(In  := IO.CycleCounter = MemCycleCounter);
	MemCycleCounter 										:= IO.CycleCounter;   	
	EventCyclecounter(
		Flag		:= TON_CycleCounter.Q AND_THEN NOT IO.WcState AND IO.InfoDataState = Tc2_EtherCAT.EC_DEVICE_STATE_OP AND Enable,
		ConfirmTrig	:= Quit OR NOT Enable AND EventCyclecounter.State <> TCEVENTSTATE_INVALID,
		MsgId		:= ,
		SourceId	:= ,
		eClass		:=,
		format		:= ,
		Text1		:= ,
		Text2		:= ,
		pText3		:= ADR(IO.DevName),
		State		=> ,
		Status		=> );	
		
	EventLogicState(
		Flag		:= IO.SafeLogicState = INVALID_SAFETY_LOGIC_STATE AND_THEN NOT IO.WcState AND IO.InfoDataState = Tc2_EtherCAT.EC_DEVICE_STATE_OP AND Enable,
		ConfirmTrig	:= Quit OR NOT Enable AND EventLogicState.State <> TCEVENTSTATE_INVALID ,
		MsgId		:= ,
		SourceId	:= ,
		eClass		:=,
		format		:= ,
		Text1		:= ,
		Text2		:= ,
		pText3		:= ADR(IO.DevName),
		State		=> ,
		Status		=> );
		
(* Read error history *********************************************)
(*	ReadDiagHist(
		Busy=> , 
		Done=> , 
		Error=> , 
		ErrorId=> , 
		Execute:= """TBD""" , 
		EcMasterDevId:= , 
		AdsAddr=> , 
		MsgInfoDiag=> , 
		DevType=> , 
		Name=> , 
		FSOEAddr=> , 
		DiagMsgSeverity=> , 
		DiagMsgTextId=> , 
		pDebugData=> , 
		DebugDataMaxId=> );	
		
	EventDiagHist(
		Flag		:= Read.msgSevyIsError AND ReadDiagHist.Done,
		ConfirmTrig	:= Quit OR NOT Enable,
		MsgId		:= ,
		SourceId	:= ,
		Class		:=,
		format		:= ,
		Text1		:= ,
		Text2		:= CONCAT('0x',DWORD_TO_HEXSTR(TO_DWORD(Read.DiagMsgTextId),4,FALSE)),
		pText3		:= ADR(IO.Name),
		State		=> ,
		Status		=> );
*)		
(* Events 11-n FB Error *******************************************)
	NoOfActiveEvents										:= 0;
	Status													:= EventInvalidCRC.Status OR EventCyclecounter.Status OR EventLogicState.status; 

	FOR i := MIN_FB TO MAX_FB 
	DO
		IF FBInfoDataDiag[i] <> 0 AND Enable
			OR EventFBError[i].State <> TCEVENTSTATE_INVALID
		THEN
			EventFBError[i](
				Flag		:= FBInfoDataDiag[i] <> 0 AND Enable,
				ConfirmTrig	:= Quit OR NOT Enable AND EventFBError[i].State <> TCEVENTSTATE_INVALID ,
				MsgId		:= ,
				SourceId	:= ,
				eClass		:= ,
				format		:= ,
				Text1		:= ,
				Text2		:= DWORD_TO_BINSTR(TO_DWORD(FBInfoDataDiag[i]),16),
				pText3		:= ADR(IO.DevName),
				State		=> );
			NoOfActiveEvents								:= NoOfActiveEvents + 1;
		END_IF	
		Status												:= Status OR EventFBError[i].Status;
	END_FOR
		

(*********************************************************)

METHOD FB_init : BOOL
VAR_INPUT
	bInitRetains : BOOL; // if TRUE, the retain variables are initialized (warm start / cold start)
	bInCopyCode : BOOL;  // if TRUE, the instance afterwards gets moved into the copy code (online change)
	
END_VAR
	FOR i := MIN_FB TO MAX_FB 
	DO
		EventFBError[i].SourceId 	:= SEL(EventFBError[i].SourceId = 0, EventFBError[i].SourceId, DEFAULT_SOURCE_ID);
		EventFBError[i].MsgId		:= TO_UINT(i + 10);
		EventFBError[i].Text1		:= INT_TO_STRING(i);	
	END_FOR
END_METHOD

PROPERTY PUBLIC sourceId : UDINT
GET
SourceId := EventLogicState.SourceId;
END_GET
SET
IF EventLogicState.SourceId <> SourceId THEN
	EventLogicState.SourceId							:= SourceId;
	EventCycleCounter.SourceId							:= SourceId;
	EventInvalidCRC.SourceId							:= SourceId;
	FOR i := MIN_FB TO MAX_FB 
	DO
		EventFBError[i].SourceId						:= SourceId;
	END_FOR
END_IF
END_SET
END_PROPERTY

END_FUNCTION_BLOCK

// POUs/Safety/Diag/SafetyPlcTerminalDiag
{attribute 'no_check'}
FUNCTION_BLOCK SafetyPlcTerminalDiag // EL6900
VAR CONSTANT
	MIN_FB													:	INT := 1;
	MAX_FB													:	INT := PARAM.SAFETY_PLC_TERM_DIAG_MAX_FB;
END_VAR                 									
VAR_INPUT               									
	Enable													:	BOOL := TRUE;	//FB will be processed as long as enable is TRUE 
	SourceId												:	UDINT := 100300;//Multisource id 
	Quit													:	BOOL;			//Resets error with rising edge 
	IO														:	EL69xx;			
END_VAR
VAR_OUTPUT
	{attribute 'displaymode':='binary'}
	Status													:	DWORD; 			//current sttus of all events
	NoOfActiveEvents										:	INT;
END_VAR
VAR (* FunctionBlock Status *)
	FBInfoDataDiag	 								AT %I*	:	ARRAY [MIN_FB..MAX_FB] OF UINT; //Safety FB diagnostic information
END_VAR
VAR (* Events/Blocks/Var internal *)
	EventInputSizeMism										: EventHandling := (SourceId := SourceId, MsgId:= 1); //Msg id 1
	EventOutputSizeMism										: EventHandling := (SourceId := SourceId, MsgId:= 2); //Msg id 2
	EventInvalidCRC											: EventHandling := (SourceId := SourceId, MsgId:= 3); //Msg id 3
	
	EventFBError											:	ARRAY [MIN_FB..MAX_FB] OF EventHandling; //MsgId from 11 to MAX_FB + 10
                        									                        	
	i														:	INT := MIN_FB;

END_VAR

(* EL6900 Safety Terminal Diag					*)
(************************************************)

(* call IO *************************************************************)
	IO();
	
(* Event 1-10 Size Mismatch ********************************************)
	EventInputSizeMism(
		Flag		:= IO.InputSizeMismatch AND Enable,
		ConfirmTrig	:= Quit OR NOT Enable AND EventInputSizeMism.State <> TCEVENTSTATE_INVALID ,
		MsgId		:= ,
		SourceId	:= ,
		eClass		:= ,
		format		:= ,
		Text1		:= ,
		Text2		:= ,
		pText3		:= ,
		State		=> );

	EventOutputSizeMism(
		Flag		:= IO.OutputSizeMismatch AND Enable,
		ConfirmTrig	:= Quit OR NOT Enable AND EventOutputSizeMism.State <> TCEVENTSTATE_INVALID ,
		MsgId		:= ,
		SourceId	:= ,
		eClass		:=,
		format		:= ,
		Text1		:= ,
		Text2		:= ,
		pText3		:= ,
		State		=> );
		
	EventInvalidCRC(
		Flag		:= IO.ProjectCRC = 0 AND_THEN NOT IO.WcState AND IO.InfoDataState = Tc2_EtherCAT.EC_DEVICE_STATE_OP AND Enable,
		ConfirmTrig	:= Quit OR NOT Enable AND EventInvalidCRC.State <> TCEVENTSTATE_INVALID ,
		MsgId		:= ,
		SourceId	:= ,
		eClass		:=,
		format		:= ,
		Text1		:= ,
		Text2		:= ,
		pText3		:= ,
		State		=> );

	
(* Events 11-n FB Error *******************************************)
	NoOfActiveEvents										:= 0;
	Status													:= EventInputSizeMism.Status OR EventOutputSizeMism.Status OR EventInvalidCRC.Status; 

	FOR i := MIN_FB TO MAX_FB 
	DO
		IF FBInfoDataDiag[i] <> 0 AND Enable
			OR EventFBError[i].State <> TCEVENTSTATE_INVALID
		THEN
			EventFBError[i](
				Flag		:= FBInfoDataDiag[i] <> 0 AND Enable,
				ConfirmTrig	:= Quit OR NOT Enable AND EventFBError[i].State <> TCEVENTSTATE_INVALID ,
				MsgId		:= ,
				SourceId	:= ,
				eClass		:= ,
				format		:= ,
				Text1		:= ,
				Text2		:= DWORD_TO_BINSTR(UINT_TO_DWORD(FBInfoDataDiag[i]),16),
				pText3		:= ,
				State		=> );
			NoOfActiveEvents								:= NoOfActiveEvents + 1;
		END_IF	
		Status												:= Status OR EventFBError[i].Status;
	END_FOR

(*********************************************************)

METHOD FB_init : BOOL
VAR_INPUT
	bInitRetains : BOOL; // if TRUE, the retain variables are initialized (warm start / cold start)
	bInCopyCode : BOOL;  // if TRUE, the instance afterwards gets moved into the copy code (online change)
END_VAR

	FOR i := MIN_FB TO MAX_FB 
	DO
		EventFBError[i].MsgId		:= TO_UINT(i + 10);
		EventFBError[i].SourceId	:= SourceId;
		EventFBError[i].Text1		:= INT_TO_STRING(i);	
		EventFBError[i].pText3		:= ADR(IO.DevName);
	END_FOR
END_METHOD

END_FUNCTION_BLOCK

// POUs/Safety/SafetyCircuit
{attribute 'no_check'}
FUNCTION_BLOCK SafetyCircuit (*  *)
VAR_INPUT  
(* periphery Outputs *)
	Demo													:	BOOL := FALSE;		//Return value TRUE = Demo mode for testing
	Enable											AT  %Q*	: 	BOOL := TRUE;		//Enable saftey circuit from PLC - map to first input of AND FB  
	Restart											AT  %Q* :	BOOL;				//Restart safety circuit  - map to restart input of estop/monitoring FB 
                                            	
(* Sequence Times *)                        	
	PT_OnOK													:	TIME := T#3S;
	PT_OnOK_2												:	TIME := T#1S500MS;
	PT_OffOK_2												:	TIME := T#1S500MS;  //be sure that then delay off time is not longer then the safety delay time
END_VAR                                     	
VAR_OUTPUT  
(* periphery Inputs *)      	
	Status													:	SAFETY_CIRCUIT_STATUS;	//Process info from EL69xx                                            	
END_VAR
VAR
	ReadyToRestart									AT  %I*	:	 BOOL; 	//TRUE when restart of safety circuit is executable
	MonOut											AT  %I*	:	 BOOL; 	//Safety estop/monitoring output direct 
	MonDelOut										AT  %I* :	 BOOL;	//Safety estop/monitoring output delay - see EStop/Monitoring FB time settings	
END_VAR
VAR
	TON_OK_1												:	TON;
	TON_OK_2												:	TON;
END_VAR

(* Safetycicrut-control with IOs and stantemachine						*)
(************************************************************************)

(* Safety circuit status *******************************************************)
IF Demo
THEN //Simulation mode 
	CASE status.state OF
	eSTATE.IDLE:	
		TON_OK_1(IN := FALSE); TON_OK_2(IN := FALSE);
		Status.RT											:= FALSE;

	eSTATE.CLEARING:
		TON_OK_2(IN := TRUE, PT := MIN(PT_OnOK_2,PT_OnOK ), Q => Status.OK_2);	
		TON_OK_1(IN := TRUE, PT := PT_OnOK , Q => Status.OK);	
		IF TON_OK_1.Q AND TON_OK_2.Q
		THEN
			Status.RT										:= TRUE;
			status.state 									:= eSTATE.IDLE;
		END_IF
	ELSE
		status.state 										:= eSTATE.CLEARING;
	END_CASE

	Status.FT												:= FALSE;
	Status.InAborting										:= status.state = eSTATE.ABORTING;
	Status.InAborted										:= status.state = eSTATE.ABORTED;
	Status.InClearing										:= status.state = eSTATE.CLEARING;
	Status.InIdle											:= status.state = eSTATE.IDLE;
	
	Status.ReadyToRestart									:= TRUE;
	Status.MonOut											:= TRUE;
	Status.MonDelOut										:= TRUE;
	
ELSE (* statemachine active mode *********************************************************)
	CASE status.state OF
	eSTATE.IDLE:
		status.RT 											:= FALSE;
		IF NOT MonOut OR NOT MonDelOut
		THEN
			TON_OK_1(IN := FALSE); TON_OK_2(IN := FALSE);
			status.state 									:= eSTATE.ABORTING;
		ELSE
			;
		END_IF

	eSTATE.ABORTING:
		IF NOT MonDelOut 
		THEN
			status.OK := status.OK_2 						:= FALSE;
			status.FT 										:= TRUE;
			status.state 									:= eSTATE.ABORTED;
		ELSIF MonOut 
		THEN
			status.FT 										:= TRUE;
			status.state 									:= eSTATE.ABORTED;
		ELSE
			TON_OK_2(IN := TRUE, PT := PT_OffOK_2);
			IF TON_OK_2.Q 
			THEN 
				status.OK_2 								:= FALSE; 
			END_IF
		END_IF

